	12000: 
		IF 	DetactSensor_B  AND FeedInSensor_B THEN
			uiExecutingStep := 12100;
		ELSIF NOT DetactSensor_B  AND FeedInSensor_B THEN
			uiExecutingStep := 12200;
		ELSIF DetactSensor_B  AND NOT FeedInSensor_B THEN
			uiExecutingStep := 12400;
		ELSIF NOT DetactSensor_B  AND NOT FeedInSensor_B THEN
			uiExecutingStep := 12400;
		END_IF
	12100: 	// two sensor on
			// Reversemotor unstill two sensor off
		ConveyorMotorB.M_MoveBackward();//('');
		tonMotorBReverse.IN :=TRUE;
		IF tonMotorBReverse.Q THEN
			tonMotorBReverse.IN :=FALSE;
			ConveyorMotorB.M_MotorStop();//('');
			uiExecutingStep :=12110;
		END_IF
		
	12110:	//wait conveyorA stop
		IF ConveyorMotorB.InStopped  THEN
			uiExecutingStep :=12120;
		END_IF
	12120:	//check two sensor
		IF DetactSensor_B OR FeedInSensor_B THEN
			_Error :=TRUE;
			strStatus :='PullOutConveyorB full box ,please remove';
		ELSE 
			uiExecutingStep :=12800;
		END_IF
		
	12200:	// FeedinSensor on
			//conveyor forward 
			FixCylinderB2.M_Extend();//('');
			IF  FixCylinderB2.InFrontPosition THEN
				ConveyorMotorB.M_MoveForward();// .M_Extend();//;//('');
				uiExecutingStep := 12840;
			END_IF		
	
	12400:	//two sensor off , need make sure no box in two sensor between 
			// Reverse motor to touch detactSensor , make sure no box 
			ConveyorMotorB.M_MoveBackward();//('');
			TON_betweenboxReverse.IN :=TRUE;
			IF TON_betweenboxReverse.Q THEN
				TON_betweenboxReverse.IN :=FALSE;
				ConveyorMotorB.M_MotorStop();//('');
				uiExecutingStep := 12410;
			END_IF
	12410:
			// wait motor stop
			IF ConveyorMotorB.InStopped  THEN
				uiExecutingStep :=12420;
			END_IF
	12420:	//check sensor
			IF DetactSensor_B THEN
				uiExecutingStep :=12430; // todo sth
			ELSIF NOT DetactSensor_B  THEN
				uiExecutingStep :=12800;
			END_IF 
	12430:	//reversemotor unstill sensor off
			ConveyorMotorB.M_MoveBackward();//('');
			TON_betweenboxReverse.IN :=TRUE;	//use to timeout 0.6s
			IF NOT DetactSensor_B THEN
				ConveyorMotorB.M_MotorStop();//('');
				uiExecutingStep :=12440;
			END_IF
			IF TON_betweenboxReverse.Q THEN
				_Error :=TRUE;
				strStatus :='PullOutConveyorB FeedIn full box ,please remove box';
			END_IF
	12440:	//wait motor stop
			IF ConveyorMotorB.InStopped  THEN
				uiExecutingStep :=12800;
			END_IF
			
	12800:	//BlockA forward and motorA forward
			BarrierCylinderB.M_Extend();//('');
			IF BarrierCylinderB.InFrontPosition THEN
				ConveyorMotorB.M_MoveForward();//;//('');
				uiExecutingStep :=12810;
			END_IF
	12810:	//wait box move in sensor and pressbox forward
			TON_PullOutTimeOut.IN 	:=TRUE;		//10S
			tonSensorDetectDelay.IN :=DetactSensor_B;		//100MS
			IF tonSensorDetectDelay.Q THEN
				tonSensorDetectDelay.IN :=FALSE;
				TON_PullOutTimeOut.IN 	:=FALSE;
				FixCylinderB2.M_Extend();//('');
				uiExecutingStep :=12820;
			END_IF
			IF TON_PullOutTimeOut.Q THEN
				_Error :=TRUE;
				strStatus :='PullOutConveyorA none box ,please refill box';
			END_IF
	12820:	//wait PressboxB2 forward & Blockbox backward 
			IF FixCylinderB2.InFrontPosition THEN
				BarrierCylinderB.M_Retract();//('');
				uiExecutingStep :=12830;
			END_IF
	12830:	//wait blockbox backward
			IF BarrierCylinderB.InRearPosition THEN
				uiExecutingStep :=12840;
			END_IF
	12840:	//delay sensor time
			TON_FeedInsensorADelay.IN := FeedInSensor_B ;
			IF TON_FeedInsensorADelay.Q THEN
				TON_FeedInsensorADelay.IN :=FALSE;
				ConveyorMotorB.M_MotorStop();//('');
				uiExecutingStep :=12850;
			END_IF
	12850:	//wait conveyor stop
			IF ConveyorMotorB.InStopped  THEN
				FixCylinderB1.M_Extend();//('');
				uiExecutingStep :=12860;
			END_IF
	12860:	//wait pressbox cylinder move
			IF FixCylinderB1.InFrontPosition THEN
				FixCylinderB1.M_Retract();//('');
				FixCylinderB2.M_Retract();//('');
				uiExecutingStep :=12870;
			END_IF
	12870:	//done
			IF FixCylinderB1.InRearPosition AND FixCylinderB2.InRearPosition THEN
				uiExecutingStep :=99000;
			END_IF
//	12000: 	
//			//check FeedinSensor & DetactSensor
//			tonMotorBReverse.IN :=TRUE;
//			ConveyorMotorb.M_MoveBackward();//('');				
//			IF tonMotorBReverse.Q  THEN
//					tonMotorBReverse.IN :=FALSE;
//					ConveyorMotorb.M_MotorStop();//('');
//					uiExecutingStep :=12005;
//			END_IF
//	12005: 	//check box leave sensor 
//			IF FeedInSensor_B OR DetactSensor_B THEN
//				_Error :=TRUE;
//				strStatus :='PullOutConveyorB full box ,please remove box';
//			ELSE
//				uiExecutingStep :=12010;
//			END_IF
	
//	12010:	//wait conveyorB stop
//			IF ConveyorMotorB.InStopped  THEN
//				uiExecutingStep := 12050;
//			END_IF
//	12050: 
//			//block forward 
//		BarrierCylinderB.M_Extend();//('');
//		IF BarrierCylinderB.In_FrontPosition THEN
//			uiExecutingStep := 12100;
//		END_IF
//	12100:	// motor forward & check detactsensor
//		ConveyorMotorB.M_Extend();//;//('');
//		TON_BoxArrivedDelay.IN := TRUE;
//		IF DetactSensor_B  THEN
//			uiExecutingStep := 12200;
//		END_IF
//		IF TON_BoxArrivedDelay.Q THEN
//			Status := 'SlideB FeedIn no box';
//			_Error := TRUE;
//		END_IF
//	12200:
//		tonSensorDetectDelay.IN :=TRUE;
//		IF tonSensorDetectDelay.Q THEN
//			FixCylinderB2.M_Extend();//('');
//			uiExecutingStep := 12300;
//		END_IF
//	12300:
//		tonSensorDetectDelay.IN :=FALSE;
//		BarrierCylinderB.M_Retract();//('');
//		IF BarrierCylinderB.In_RearPosition THEN
//			uiExecutingStep := 12400;
//		END_IF
//	12400:
//		TON_BoxArrivedDelay.IN := TRUE;
//		IF FeedInSensor_B THEN
//			ConveyorMotorB.M_MotorStop();//('');
//			uiExecutingStep := 12500;
//		END_IF
//		IF TON_BoxArrivedDelay.Q THEN
//			Status := 'SlideB FeedIn no box';
//			_Error := TRUE;
//		END_IF
//	12500:
//		FixCylinderB1.M_Extend();//('');
//		uiExecutingStep := 12510;
//	12510:
//		TON_BarryDelay.IN := TRUE;
//		IF TON_BarryDelay.Q THEN
//			FixCylinderB1.M_Retract();//('');
//			FixCylinderB2.M_Retract();//('');
//			uiExecutingStep := 99000;
//		END_IF
{endregion}

	50000:	//SlideA FeedIn Ext Resume step
			FixCylinderA1.M_Retract();
			FixCylinderA2.M_Retract();
			BarrierCylinderA.M_Retract();
			ConveyorMotorA.M_MotorStop();
			TON_PullOutTimeOut.IN :=FALSE;
			TON_betweenboxReverse.IN :=FALSE;
			IF FixCylinderA1.InRearPosition AND 
				FixCylinderA2.InRearPosition AND 
				BarrierCylinderA.InRearPosition AND 
				ConveyorMotorA.InStopped THEN
				_Abort :=TRUE;
			END_IF
			
    99000:
        TON_MotorStopDelay.IN := FALSE;
        _Executed             := TRUE;

END_CASE

IF _Executed THEN
    eState := STATE_DONE;
ELSIF NOT Execute THEN
    eState := STATE_RESETTING;
ELSIF _Abort OR Abort THEN
    eState := STATE_ABORTING;
ELSIF _Error THEN
	eState:=STATE_ERROR;	
END_IF
END_METHOD

METHOD  M_STATE_RESETTING
VAR_INPUT
END_VAR
CASE uiResettingStep OF
	0:
		FixCylinderA1.M_Retract();// .M_Retract();//('Resetting');
		FixCylinderA2.M_Retract();//('Resetting');
		FixCylinderB1.M_Retract();//('Resetting');
		FixCylinderB2.M_Retract();//('Resetting');
		BarrierCylinderA.M_Retract();//('Resetting');
		BarrierCylinderB.M_Retract();//('Resetting');
		uiResettingStep := 100;
	100:
		IF FixCylinderA1.InRearPosition AND
			FixCylinderA2.InRearPosition AND
			FixCylinderB1.InRearPosition AND
			FixCylinderB2.InRearPosition AND
			BarrierCylinderA.InRearPosition AND 
			BarrierCylinderB.InRearPosition THEN
			uiResettingStep := 200;
		END_IF
	200:
		ConveyorMotorA.M_MotorStop();// .M_StopMotor('Resetting');
		ConveyorMotorB.M_MotorStop();
		uiResettingStep := 300;
	300:
		IF ConveyorMotorA.InStopped AND 
			ConveyorMotorB.InStopped THEN
		//	DAS.fbStorageArea.M_InactivePulloutConveyorInternCtrl();
			uiResettingStep := 9000;
		END_IF
	9000:
		_Error :=false;
		 Error :=false;
		_ResetCompleted := TRUE;
END_CASE
IF _ResetCompleted THEN
	eState := STATE_DORMANT;
END_IF
END_METHOD

END_FUNCTION_BLOCK

// ---- Library/20_MachineUnits/22_AllocateArea/Service/FB_PullOutConveyorBtnCtrl.TcPOU
FUNCTION_BLOCK FB_PullOutConveyorBtnCtrl 
VAR_INPUT
	Input	:REFERENCE TO ST_InputTable;
	Output	:REFERENCE TO ST_OutputTable;
//	ConveyorMotorA :REFERENCE TO FB_Motor;
//	ConveyorMotorB :REFERENCE TO FB_Motor;
	Motor	:REFERENCE TO UNI_MotorList;
	
	
	bPullOutConveyorExecute	:BOOL;
	bPullOutConveyorDone	:BOOL;
	bPullOutConveyorBusy	:BOOL;
	StroageRegionMode :E_UnitMode ;
END_VAR
VAR_OUTPUT
	PullOutConveyorState :E_PullOutConveyorState;
END_VAR
VAR
	ExecutingStep	:E_PullOutConveyorState;
	bReferenceComponetIsRefed :BOOL;
	Forward_EdgeDetect	:FB_EdgeDetect;
	Backward_EdgeDetect	:FB_EdgeDetect;
END_VAR

clcUpdate();
Forward_EdgeDetect(xInput:=Input.bPullOutCV_FwdPb);
Backward_EdgeDetect(xInput :=Input.bPullOutCV_RevPb);
//IF __ISVALIDREF(BtnMoveForward) AND
//	__ISVALIDREF(BtnMoveReverse) AND
//	__ISVALIDREF(ConveyorMotorA) AND
//	__ISVALIDREF(ConveyorMotorB) THEN
	
//	bReferenceComponetIsRefed :=TRUE;
//END_IF

//IF bReferenceComponetIsRefed THEN
//	clcUpdate();
//END_IF

METHOD PRIVATE clcUpdate : BOOL
VAR_INPUT
END_VAR

CASE ExecutingStep OF
	E_PullOutConveyorState.idle:
	;
	
	E_PullOutConveyorState.AutoMode:
		M_TurnOff();
		M_TurnOff();
			IF bPullOutConveyorDone AND 
				NOT bPullOutConveyorExecute AND 
				NOT (StroageRegionMode = E_MachineMode.AUTO)  THEN
				ExecutingStep := E_PullOutConveyorState.Free;
			END_IF
	
	E_PullOutConveyorState.Free:
		M_TurnOn();
		M_TurnOn();
		IF NOT (StroageRegionMode = E_UnitMode.AUTO) AND 
				(StroageRegionMode = E_UnitMode.MANUAL) THEN
//			IF BtnMoveReverse.P_ButtonState AND BtnMoveForward.P_ButtonState THEN
			IF Input.bPullOutCV_FwdPb AND Input.bPullOutCV_RevPb THEN
//				ConveyorMotorA.M_StopMotor('');
//				ConveyorMotorB.M_StopMotor('');
				Motor.List.PullOutCV_A.M_MotorStop();
				Motor.List.PullOutCV_B.M_MotorStop();
					ELSIF Forward_EdgeDetect.xFallingEdge THEN 
						Motor.List.PullOutCV_A.M_MotorStop();
						Motor.List.PullOutCV_B.M_MotorStop();
					ELSIF Backward_EdgeDetect.xFallingEdge THEN
						Motor.List.PullOutCV_A.M_MotorStop();
						Motor.List.PullOutCV_B.M_MotorStop();
					ELSIF Input.bPullOutCV_RevPb THEN
							Motor.List.PullOutCV_A.M_MoveBackward();
							Motor.List.PullOutCV_B.M_MoveBackward();
					ELSIF Input.bPullOutCV_FwdPb  THEN
							Motor.List.PullOutCV_A.M_MoveForward();
							Motor.List.PullOutCV_B.M_MoveForward();					
			END_IF
		END_IF
END_CASE

IF (bPullOutConveyorExecute AND bPullOutConveyorBusy ) OR (StroageRegionMode = E_UnitMode.AUTO)  THEN
	ExecutingStep := E_PullOutConveyorState.AutoMode;
ELSE
	ExecutingStep := E_PullOutConveyorState.Free;
END_IF

PullOutConveyorState:=ExecutingStep;
END_METHOD

METHOD PRIVATE M_TurnOff : BOOL
VAR_INPUT
END_VAR
Output.bPullOutCV_FwdPbLamp:=FALSE;
Output.bPullOutCV_RevPbLamp:=FALSE;
END_METHOD

METHOD PRIVATE M_TurnOn : BOOL
VAR_INPUT
END_VAR
Output.bPullOutCV_FwdPbLamp:=TRUE;
Output.bPullOutCV_RevPbLamp:=TRUE;
END_METHOD

END_FUNCTION_BLOCK

// ---- Library/20_MachineUnits/22_AllocateArea/Service/FB_AllocateRobotNeedlingMove.TcPOU
FUNCTION_BLOCK FB_AllocateRobotNeedlingMove EXTENDS FB_ActionBasic
VAR_INPUT
    xExecute      : BOOL;
    xAbort        : BOOL;
    TimeOut  : LREAL := 30; // Unit : s
	MovingInfo	: ST_AllocateRobotNeedlingMoveInfo;
END_VAR
VAR_OUTPUT
    xAborted : BOOL;
    iErrorID : INT;
    ErrorMsg : T_MaxString;
END_VAR
VAR
    StateBehavior   : CBML.ETrigATo;
    uiCyclicStep    : UINT := 0;
    uiIndexLoop     : UINT;
	Coordinate		:st_Coordinate;
	fbExecuteEdgeDetect :FB_EdgeDetect;
END_VAR

THIS^.IBehaviourModel := StateBehavior;
StateBehavior(xExecute := xExecute,
              xAbort := xAbort OR fbExecuteEdgeDetect.xFallingEdge,
              udiTimeOut := LREAL_TO_UDINT( TimeOut*1000000),
              xDone => xDone,
              xBusy => xBusy,
              xError => xError,			  
              xAborted => xAborted);			  

			  
//Make sure that C# turns off execute to shut down the service
fbExecuteEdgeDetect(xInput :=xExecute);

//Error Msg
iErrorID := StateBehavior._model.iErrorID;
ErrorMsg := M_GetErrorMsg(xErrorID := iErrorID);

METHOD CleanupAction
VAR_INPUT
    xAbortProposed : BOOL;
    iErrorIDProposed: INT;
END_VAR
VAR_OUTPUT
    xComplete : BOOL := TRUE;
    xAbort: BOOL := xAbortProposed;
 	iErrorID : INT := iErrorIDProposed;
END_VAR
uiCyclicStep := 0;
END_METHOD

METHOD CyclicAction
VAR_INPUT
    itfTimingController : CBML.ITimingController;
END_VAR
VAR_OUTPUT
    xComplete : BOOL := TRUE;
    iErrorID : INT := 0;
END_VAR
VAR_INST
	
END_VAR

VAR
		bAxesCheck 		: BOOL;
	
	
END_VAR
xComplete := FALSE;

	IF arAxisCtrl_gb[AxisNo.Allocate_X].Admin.Axis.Status.Error OR
		arAxisCtrl_gb[AxisNo.Allocate_Y].Admin.Axis.Status.Error THEN
		iErrorID :=3;
	END_IF

CASE uiCyclicStep OF
    0:
		
			uiCyclicStep:=100;
		
		
	100:
			arAxisCtrl_gb[AxisNo.Allocate_X].PosMode.Position:=Coordinate.X;
			arAxisCtrl_gb[AxisNo.Allocate_Y].PosMode.Position:=Coordinate.Y;	
		
			IF arAxisCtrl_gb[AxisNo.Allocate_X].Admin.Axis.Status.Moving OR
			   arAxisCtrl_gb[AxisNo.Allocate_Y].Admin.Axis.Status.Moving OR
			   arAxisStatus_gb[AxisNo.Allocate_X].Admin._OpModeAck=E_AXIS_MODE.ModePosAbs OR
			   arAxisStatus_gb[AxisNo.Allocate_y].Admin._OpModeAck=E_AXIS_MODE.ModePosAbs THEN
			   uiCyclicStep:=200;
			END_IF
			
	200:
			bAxesCheck := TRUE;

		bAxesCheck := bAxesCheck AND	 arAxisStatus_gb[AxisNo.Allocate_x].Admin.CmdDone ;
		bAxesCheck := bAxesCheck AND	 arAxisStatus_gb[AxisNo.Allocate_y].Admin.CmdDone ;	
	
		IF bAxesCheck THEN
			 uiCyclicStep:=600;
		END_IF
	600:
		
		xComplete := TRUE;
END_CASE
END_METHOD

METHOD ExitAction
VAR_INPUT
    xAfterCleanup : BOOL;
    xInCopyCode : BOOL;
END_VAR
END_METHOD

METHOD PRIVATE M_CheckCommand : BOOL
VAR_INPUT
END_VAR
VAR_OUTPUT
	iErrorID	 : INT :=0 ;
END_VAR
VAR
	
END_VAR
IF MovingInfo.Box<0 OR MovingInfo.Box >1 OR MovingInfo.Clip<0 OR MovingInfo.Clip>3 OR MovingInfo.NeedleLocation<0 OR MovingInfo.NeedleLocation>49 THEN
	iErrorID :=2;
	M_CheckCommand := FALSE;
	RETURN;
END_IF

IF MovingInfo.Area = 'T' THEN
		
	FUN_GetNeedleCoordinates(uiLocation :=1 ,
							 uiBox:=MovingInfo.Box,
							 uiClip:=MovingInfo.Clip,
							 uiNeedleLocation:=MovingInfo.NeedleLocation,
							 NeedleCoordinate=>Coordinate);
	IF MovingInfo.Box = 1 AND (MovingInfo.Clip = 2 OR MovingInfo.Clip = 3) THEN
		M_CheckCommand := FALSE;
		iErrorID :=2;
		RETURN;
	END_IF
	IF MovingInfo.Box = 2 AND (MovingInfo.Clip = 0 OR MovingInfo.Clip = 1) THEN
		M_CheckCommand :=FALSE;
		iErrorID :=2;
		RETURN;
	END_IF
	
ELSIF 	

	MovingInfo.Area = 'Q' THEN
	FUN_GetNeedleCoordinates(uiLocation :=0 ,
							 uiBox:=MovingInfo.Box,
							 uiClip:=MovingInfo.Clip,
							 uiNeedleLocation:=MovingInfo.NeedleLocation,
							 NeedleCoordinate=>Coordinate);
	

ELSE
	iErrorID :=2;
	M_CheckCommand := FALSE;
	RETURN;
END_IF

M_CheckCommand:=TRUE;
END_METHOD

METHOD M_GetErrorMsg : T_MaxString
VAR_INPUT
	xErrorID: INT;
END_VAR

VAR
	
END_VAR
CASE xErrorID OF
	0:
		M_GetErrorMsg := 'No Error';
	1:
		M_GetErrorMsg := 'Action time out';
	2:
		M_GetErrorMsg := 'Wrong command';
	3:
		M_GetErrorMsg := 'Servo axis error';
//	4:
//		M_GetErrorMsg := 'Axis roundbelt not ready has Error';
//	5:
//		M_GetErrorMsg := 'Cylinder not ready has Error';
//	6:
//		M_GetErrorMsg := 'Axis RoundBelt has Error';
//	7:
//		M_GetErrorMsg := 'ChargeZone_Plug has Error';
//	8:
//		M_GetErrorMsg := 'TransmitCVZone_Plug has Error';
//	9:
//		M_GetErrorMsg := 'WorkZone_Plug has Error';
//	10:
//		M_GetErrorMsg := 'WorkZone_Press has Error';
END_CASE
END_METHOD

METHOD PRIVATE M_ResetAxes : BOOL
VAR_INPUT
END_VAR
VAR
	bAxesCheck :BOOL;
END_VAR
		bAxesCheck :=TRUE;
		IF arAxisCtrl_gb[AxisNo.Allocate_X].Admin.Axis.Status.Error THEN
			arAxisCtrl_gb[AxisNo.Allocate_X].Admin.ClearError:=TRUE;			
			ELSE
			arAxisCtrl_gb[AxisNo.Allocate_X].Admin.ClearError:=FALSE;	
		END_IF
		IF arAxisCtrl_gb[AxisNo.Allocate_Y].Admin.Axis.Status.Error THEN
			arAxisCtrl_gb[AxisNo.Allocate_Y].Admin.ClearError:=TRUE;			
			ELSE
			arAxisCtrl_gb[AxisNo.Allocate_Y].Admin.ClearError:=FALSE;	
		END_IF
		bAxesCheck := bAxesCheck AND NOT arAxisCtrl_gb[AxisNo.Allocate_X].Admin.ClearError ;
		bAxesCheck := bAxesCheck AND NOT arAxisCtrl_gb[AxisNo.Allocate_X].Admin.ClearError ;
		
		M_ResetAxes := bAxesCheck;
END_METHOD

METHOD ResetAction
VAR_OUTPUT
    xComplete : BOOL := TRUE;
END_VAR
uiCyclicStep := 0;
END_METHOD

METHOD StartAction
VAR_OUTPUT
    xComplete : BOOL := TRUE;
	iErrorID : INT := 0;
END_VAR
xComplete := FALSE;
uiCyclicStep := 0;

IF M_CheckCommand(iErrorID=>iErrorID) AND M_ResetAxes() THEN
	xComplete := TRUE;
END_IF
END_METHOD

END_FUNCTION_BLOCK

// ---- Library/20_MachineUnits/22_AllocateArea/Duts/F_Even.TcPOU
FUNCTION F_Even : BOOL
VAR_INPUT
	uiNumber		: UINT;
END_VAR
VAR
END_VAR

F_Even := uiNumber MOD 2 = 0;

END_FUNCTION

// ---- Library/20_MachineUnits/21_StorageArea/FB_StorageArea.TcPOU
FUNCTION_BLOCK FB_StorageArea EXTENDS FB_ModeBase_V2 IMPLEMENTS I_UnitState
VAR_INPUT
    FanucRobot : REFERENCE TO FB_FanucRobot_Basic;
    Service    : REFERENCE TO ST_StorageService;

    Cylinder : REFERENCE TO UNI_CylinderList;
    Motor    : REFERENCE TO UNI_MotorList;

    Input            : REFERENCE TO ST_InputTable;
    OutPut           : REFERENCE TO ST_OutputTable;
    Reset            : REFERENCE TO BOOL;
	Stop :  REFERENCE TO BOOL;
	bStopMem :  REFERENCE TO BOOL;
    WheelhouseSensor : REFERENCE TO UNI_HMI_WheelHouseInput;
    CurrentData      : ST_SetupPara;
END_VAR
VAR_OUTPUT
	RobotResetCMD :BOOL;
	Homed : BOOL;
END_VAR
VAR
    // Service
    fbFeedInEmptyBoxWithRobot           : FB_FeedInEmptyBoxWithRobot;
    fbReloadRoundBeltBoxWithRobot       : FB_ReloadRoundBeltBoxWithRobot;
    fbRobotRegionMove_AllocatedConveyor : FB_RobotRegionMove_AllocatedConveyor;
    fbRobotRegionMove_BufferArea        : FB_RobotRegionMove_BufferArea;
    fbRobotRegionMove_FeedInConveyor    : FB_RobotRegionMove_FeedInConveyor;
    fbRobotRegionMove_PullOutConveyor   : FB_RobotRegionMove_PullOutConveyor;
    fbRobotRegionMove_RoundBelt         : FB_RobotRegionMove_RoundBelt;
    fbRobotAbsMove                      : FB_RobotAbsMove;
    fbWareHouseWithRobotMove            : FB_WareHouseWithRobotMove;
	fbStorageHoming 					: FB_StorageHoming;
	//UpCV
    _fbDaimeterMovement   			: FB_DiameterMovement; //UpCV Internal use
    fbUpperFeedInConveyor 			: FB_UpperFeedInConveyor;
	fbAddBoxes                      : FB_AddBoxes_v2;
	fbBoxSupplyCtrl					: FB_BoxSupplyCtrl;
    RackState                       : E_RackState;
    
    // Pullout
    fbPullOutConveyorAction         : FB_PullOutConveyorAction;
    AutoPullout_Ctrl                : ST_AutoPullOutConveyorCommand;
    AutoPullout_Status              : ST_AutoPullOutConveyorSatus;
    AutoPullout_Info                : ST_PullOutConveyorInfo;
    bPulloutConveyorInternCtrl      : BOOL := FALSE;
    AutoMode_PulloutConveyor_Intern : ST_AutoPullOutConveyor; // Pullout conveyor inter
    

    // Robot abs move
    RobotAbsMoveAuto_Ctrl   : st_RobotAbsMove_Ctrl;
    RobotAbsMoveAuto_Status : st_RobotAbsMove_Status;
    RobotAbsMoveAuto_Info   : st_AutoSixAxisAbsMoveParameter;
    // Warehouse
	fbWarehouse           : FB_WareHouse;
    //========= Auto Mode Robot Warehouse Move =================
    RobotWarehouseMoveAuto_Ctrl   : st_RobotWarehouseMove_Ctrl;
    RobotWarehouseMoveAuto_Status : st_RobotWarehouseMove_Status;

    _RobotWarehouseMoveAuto_Ctrl   : st_RobotWarehouseMove_Ctrl;
    _RobotWarehouseMoveAuto_Status : st_RobotWarehouseMove_Status;

    RobotWarehouseMoveAuto_internal_Ctrl   : st_RobotWarehouseMove_Ctrl;
    RobotWarehouseMoveAuto_internal_Status : st_RobotWarehouseMove_Status;
    bWarehouseMoveInternalAccess           : BOOL := FALSE;
	// Storage homing
	StorageHoming_Execute : BOOL;
	StorageHoming_Reset : BOOL;
	StorageHoming_Abort : BOOL;
	StorageHoming_Busy : BOOL;
	StorageHoming_Done : BOOL;
	StorageHoming_Error : BOOL;
END_VAR

SUPER^();

IF __ISVALIDREF(PackTag) THEN
    eModeCommand := PackTag.Command.UnitMode;
    eStateCommand := PackTag.Command.CntrlCmd;
ELSE
    RETURN;
END_IF

ACTION A00_Service:
fbFeedInEmptyBoxWithRobot(Execute    := service.AutoMode_FeedInEmptyBoxWithRobot.Command.Execute,
                          Abort      := service.AutoMode_FeedInEmptyBoxWithRobot.Command.Abort,
                          Reset      := Reset,
                          ObjectName := 'FeedInEmptyBox with robot',
                          Busy       => service.AutoMode_FeedInEmptyBoxWithRobot.Status.Busy,
                          Done       => service.AutoMode_FeedInEmptyBoxWithRobot.Status.Done,
                          Aborted    =>,
                          Error      => service.AutoMode_FeedInEmptyBoxWithRobot.Status.Error,
                          ErrorID    =>,
                          Status     => service.AutoMode_FeedInEmptyBoxWithRobot.Status.Status,
                          UniqueErrorCode   =>,
                          Robot      := FanucRobot,
                          WareHouse  := fbWarehouse,
                          Input      := Input,
                          DiffSizeCV := Motor.List.TransmitDifferentSideCV,
						  SameSizeCV := Motor.List.TransmitSameSideCV,
                          Info := Service.AutoMode_FeedInEmptyBoxWithRobot.Info,
                          Stop := bStopMem);

fbRobotRegionMove_BufferArea(Execute	:= Service.AutoMode_RobotRegionMove_BufferArea.Command.Execute,
                             Abort 		:= Service.AutoMode_RobotRegionMove_BufferArea.Command.Abort,
                             Reset 		:= Reset,
                             ObjectName	:= 'RobotRegionMove_BufferArea',
                             Busy    => Service.AutoMode_RobotRegionMove_BufferArea.Status.Busy,
                             Done    => Service.AutoMode_RobotRegionMove_BufferArea.Status.Done,
                             Aborted =>,
                             Error   => Service.AutoMode_RobotRegionMove_BufferArea.Status.Error,
                             ErrorID =>,
                             Status  => Service.AutoMode_RobotRegionMove_BufferArea.Status.Status,
							 UniqueErrorCode	=>,
                             Robot 	:= FanucRobot,
                             Info 	:= Service.AutoMode_RobotRegionMove_BufferArea.Info,
                             Stop 	:= bStopMem);

fbPullOutConveyorAction(Execute          := (*AutoPullout_Ctrl.Execute*) ,
                        Abort            := AutoPullout_Ctrl.Abort,
                        Reset            := Reset,
                        ObjectName       := 'fbPullOutConveyorAction',
                        Busy             => AutoPullout_Status.Busy,
                        Done             => AutoPullout_Status.Done,
                        Aborted          =>,
                        Error            => AutoPullout_Status.Error,
                        ErrorID          =>,
                        Status           => AutoPullout_Status.Status,
                        UniqueErrorCode  =>,
                        FixCylinderA1    := Cylinder.List.fbPullOutCV_AsidePress1,
                        FixCylinderA2    := Cylinder.List.fbPullOutCV_AsidePress2,
                        FixCylinderB1    := Cylinder.List.fbPullOutCV_BsidePress1,
                        FixCylinderB2    := Cylinder.List.fbPullOutCV_BsidePress2,
                        BarrierCylinderA := Cylinder.List.fbPullOutCV_AsideBlock,
                        BarrierCylinderB := Cylinder.List.fbPullOutCV_BsideBlock,
                        ConveyorMotorA   := Motor.List.PullOutCV_A,
                        ConveyorMotorB   := Motor.List.PullOutCV_B,
                        INPUT            := INPUT,
                        PullOutInfo      := AutoPullout_Info);

fbUpperFeedInConveyor(Execute             := Service.AutoMode_UpperFeedInConveyor.Command.Execute,
                      Abort               := Service.AutoMode_UpperFeedInConveyor.Command.Abort,
                      Reset               := Reset,
                      ObjectName          := 'Storage_UpperFeedInConveyor',
                      Busy                => Service.AutoMode_UpperFeedInConveyor.Status.Busy,
                      Done                => Service.AutoMode_UpperFeedInConveyor.Status.Done,
                      Aborted             =>,
                      Error               => Service.AutoMode_UpperFeedInConveyor.Status.Error,
                      ErrorID             =>,
                      Status              =>,
                      UniqueErrorCode     =>,
                      _fbDiameterMovement := THIS^._fbDaimeterMovement,
                      Cylinder            := Cylinder,
                      Motor               := Motor,
                      Input               := Input,
                      OutPut              := OutPut,
                      Info                := Service.AutoMode_UpperFeedInConveyor.Info,
                      AddingBox           :=,
                      FeedBack            => Service.AutoMode_UpperFeedInConveyor.FeedBack,
					  _bForceUpperCV_Use   =>	);

_fbDaimeterMovement(Execute         :=,
                    Abort           :=,
                    Reset           :=,
                    ObjectName      :=,
                    Busy            =>,
                    Done            =>,
                    Aborted         =>,
                    Error           =>,
                    ErrorID         =>,
                    Status          =>,
                    UniqueErrorCode =>,
                    bContinue       :=,
                    Cylinder        := Cylinder,
                    PickDone        =>);

fbWarehouse(Motors           := Motor,
            WheelhouseSensor := WheelhouseSensor);

fbAddBoxes(Execute                   := Service.AutoMode_AddBoxes.Command.Execute,
           Abort                     := Service.AutoMode_AddBoxes.Command.Abort,
           Reset                     := Reset,
           ObjectName                := 'Storage_AddBoxes',
           Busy                      => Service.AutoMode_AddBoxes.Status.Busy,
           Done                      => Service.AutoMode_AddBoxes.Status.Done,
           Aborted                   =>,
           Error                     => Service.AutoMode_AddBoxes.Status.Error,
           ErrorID                   =>,
           Status                    =>,
           UniqueErrorCode           =>,
           Cylinder                  := Cylinder,
           Motor                     := Motor,
           Input                     := Input,
           OutPut                    := OutPut,
           CurrentData               := CurrentData,
           ERackState                := RackState,
           bClearInterventionRequest :=,
           InterventionRequest       => Service.AutoMode_AddBoxes.Status.InterventionRequest,
           FeedingBoxes              => Service.AutoMode_AddBoxes.Status.FeedingBoxes,
			_bForceUpperCV_Use 		:= fbUpperFeedInConveyor._bForceUpperCV_Use);

fbBoxSupplyCtrl(Execute           := TRUE,
                Abort             :=,
                Reset             :=reset,
                ObjectName        :=,
                Busy              =>,
                Done              =>,
                Aborted           =>,
                Error             =>,
                ErrorID           =>,
                Status            =>,
                UniqueErrorCode   =>,
                Cylinder          := Cylinder,
                CurrentData       := CurrentData,
                Input             := Input,
                Output            := OutPut,
                StroageRegionMode := eModeCurrent,
                bAddsBoxRequest   := Service.AutoMode_AddBoxes.Status.InterventionRequest,
                AddBoxes_Status   := Service.AutoMode_AddBoxes.Status,
                AddBoxes_Ctrl     := Service.AutoMode_AddBoxes.Command,
				AxisRackMotorBTNHomeRequest=>,
                RackState         => RackState);

fbRobotRegionMove_FeedInConveyor(Execute 	:= Service.AutoMode_RobotRegionMove_FeedInConveyor.Command.Execute,
                                 Abort 		:= Service.AutoMode_RobotRegionMove_FeedInConveyor.Command.Abort,
                                 Reset      := Reset,
                                 ObjectName := 'Storage Robot FeedIn CV',
                                 Busy       => Service.AutoMode_RobotRegionMove_FeedInConveyor.Status.Busy,
                                 Done 		=> Service.AutoMode_RobotRegionMove_FeedInConveyor.Status.Done,
                                 Aborted	=>,
                                 Error   	=> Service.AutoMode_RobotRegionMove_FeedInConveyor.Status.Error,
                                 ErrorID 	=>,
                                 Status  	=> Service.AutoMode_RobotRegionMove_FeedInConveyor.Status.Status,
                                 UniqueErrorCode =>,
                                 Robot           := FanucRobot,
                                 LowerConveyor   := Motor.List.LowCV,
                                 Input           := Input,
                                 //								 F1SensorOfUpperConveyor :=Input.bUpCV_BoxArrived_Sensor,
                                 //								 Input.bUpCV_Block1Detect_Sensor := Input.bUpCV_Block1Detect_Sensor ,
                                 Info := Service.AutoMode_RobotRegionMove_FeedInConveyor.Info,
                                 Stop :=bStopMem);

fbRobotRegionMove_AllocatedConveyor(Execute 	:= Service.AutoMode_RobotRegionMove_AllocatedConveyor.Command.Execute,
                                    Abort 		:= Service.AutoMode_RobotRegionMove_AllocatedConveyor.Command.Abort,
                                    Reset  		:= Reset,
                                    ObjectName 	:= ' Storage Robot Transmit CV',
                                    Busy       	=> Service.AutoMode_RobotRegionMove_AllocatedConveyor.Status.Busy,
                                    Done 		=> Service.AutoMode_RobotRegionMove_AllocatedConveyor.Status.Done,
                                    Aborted 	=>,
                                    Error   	=> Service.AutoMode_RobotRegionMove_AllocatedConveyor.Status.Error,
                                    ErrorID 	=>,
                                    Status  	=> Service.AutoMode_RobotRegionMove_AllocatedConveyor.Status.Status,
                                    UniqueErrorCode =>,
                                    Robot           := FanucRobot,
                                    DifferenceCV    := Motor.List.TransmitDifferentSideCV,
                                    SamesizeCV      := Motor.List.TransmitSameSideCV,
                                    cylinder        := Cylinder,
                                    //	SameSizeFullSensor:= , 
                                    Input := Input,
                                    Info := service.AutoMode_RobotRegionMove_AllocatedConveyor.Info,
                                    Stop :=bStopMem);


fbRobotRegionMove_PullOutConveyor(Execute 	:=Service.AutoMode_RobotRegionMove_PullOutConveyor.Command.Execute,
                                  Abort 	:=Service.AutoMode_RobotRegionMove_PullOutConveyor.Command.Abort,
                                  Reset     := Reset,
                                  ObjectName:= 'Storage Robot PulloutCV',
                                  Busy      => Service.AutoMode_RobotRegionMove_PullOutConveyor.Status.Busy,
                                  Done 		=> Service.AutoMode_RobotRegionMove_PullOutConveyor.Status.Done,
                                  Aborted 	=>,
                                  Error   	=> Service.AutoMode_RobotRegionMove_PullOutConveyor.Status.Error,
                                  ErrorID 	=>,
                                  Status  	=> Service.AutoMode_RobotRegionMove_PullOutConveyor.Status.Status,
                                  UniqueErrorCode =>,
                                  Robot           := FanucRobot,
                                  PullOutConveyor := fbPullOutConveyorAction,
                                  Info := Service.AutoMode_RobotRegionMove_PullOutConveyor.Info,
                                  Stop :=bStopMem);

fbRobotAbsMove(Execute         := Service.AutoMode_RobotAbsMove.HandShake.Execute,
               Abort           :=,
               Reset           := Reset,
               ObjectName      := 'Storage robot abs move',
               Busy            => Service.AutoMode_RobotAbsMove.HandShake.Busy,
               Done            => Service.AutoMode_RobotAbsMove.HandShake.Done,
               Aborted         =>,
               Error           => Service.AutoMode_RobotAbsMove.HandShake.Error,
               ErrorID         =>,
               Status          =>,
               UniqueErrorCode =>,
               Robot           := FanucRobot,
               LowerConveyor   := Motor.List.LowCV,
               Info            := Service.AutoMode_RobotAbsMove,
               Input 		:= Input,
               Stop :=bStopMem);

fbRobotRegionMove_RoundBelt(Execute := Service.AutoMode_RobotRegionMove_RoundBelt.Command.Execute,
                            Abort   := Service.AutoMode_RobotRegionMove_RoundBelt.Command.Abort,
                            Reset   := Reset,
                            ObjectName:= 'Storage robot  RegionMove roundbelt',
                            Busy    => Service.AutoMode_RobotRegionMove_RoundBelt.Status.Busy,
                            Done    => Service.AutoMode_RobotRegionMove_RoundBelt.Status.Done,
                            Aborted =>,
                            Error   => Service.AutoMode_RobotRegionMove_RoundBelt.Status.Error,
                            ErrorID =>,
                            Status 	=> Service.AutoMode_RobotRegionMove_RoundBelt.Status.Status,
                            UniqueErrorCode =>,
                            Robot 		:= FanucRobot,
                            RoundBelt 	:= DAS_CoreSys.MachineControl.fbAllocateArea.RoundBeltControl,
							Input 		:= Input,
                            Info 		:= Service.AutoMode_RobotRegionMove_RoundBelt.Info,
                            Stop 		:=bStopMem);

fbReloadRoundBeltBoxWithRobot(Execute	:= Service.AutoMode_ReloadRoundBeltBoxWithRobot.Command.Execute,
                              Abort 	:= Service.AutoMode_ReloadRoundBeltBoxWithRobot.Command.Abort,
                              Reset 	:= Reset,
                              ObjectName:= 'Storage robot reload roundbelt',
                              Busy    => Service.AutoMode_ReloadRoundBeltBoxWithRobot.Status.Busy,
                              Done    => Service.AutoMode_ReloadRoundBeltBoxWithRobot.Status.Done,
                              Aborted =>,
                              Error   => Service.AutoMode_ReloadRoundBeltBoxWithRobot.Status.Error,
                              ErrorID =>,
                              Status  => Service.AutoMode_ReloadRoundBeltBoxWithRobot.Status.Status,
                              UniqueErrorCode =>,
                              Robot 	:= FanucRobot,
                              RoundBelt := DAS_CoreSys.MachineControl.fbAllocateArea.RoundBeltControl,
                              WareHouse := fbWarehouse,
                              Input 	:= Input,
                              Info 		:= Service.AutoMode_ReloadRoundBeltBoxWithRobot.Info,
                              Stop 		:= bStopMem);
//============================ Auto Mode Robot Warehouse Move =============================
IF NOT bWarehouseMoveInternalAccess THEN
    _RobotWarehouseMoveAuto_Ctrl := RobotWarehouseMoveAuto_Ctrl;
    RobotWarehouseMoveAuto_Status := _RobotWarehouseMoveAuto_Status;
ELSE
    _RobotWarehouseMoveAuto_Ctrl := RobotWarehouseMoveAuto_internal_Ctrl;
    RobotWarehouseMoveAuto_internal_Status := _RobotWarehouseMoveAuto_Status;
END_IF

(*M_RobotWarehouseMove(
        bExecute  := Service.AutoMode_RobotWarehouseMove.HandShake.Execute,
        bReset    := Service.AutoMode_RobotWarehouseMove.HandShake.Reset,
        bAbort    := FALSE,
        bOccupied := FALSE,
        eMode     := E_MachineMode.Auto,
        bBusy     => Service.AutoMode_RobotWarehouseMove.HandShake.Busy,
        bDone     => Service.AutoMode_RobotWarehouseMove.HandShake.Done,
        bError    => Service.AutoMode_RobotWarehouseMove.HandShake.Error);*)
fbWareHouseWithRobotMove(
	Execute:= Service.AutoMode_WarehouseMotoWithRobotMove.HandShake.Execute, 
	Abort:= , 
	Reset:= Reset, 
	ObjectName:= 'storage Robot Warehouse move', 
	Busy=> Service.AutoMode_WarehouseMotoWithRobotMove.HandShake.Busy, 
	Done=> Service.AutoMode_WarehouseMotoWithRobotMove.HandShake.Done, 
	Aborted=> , 
	Error=> Service.AutoMode_WarehouseMotoWithRobotMove.HandShake.Error, 
	ErrorID=> , 
	Status=> , 
	UniqueErrorCode=> , 
	Robot:= FanucRobot, 
	WareHouse:= fbWarehouse, 
	Info:= Service.AutoMode_WarehouseMotoWithRobotMove, 
	Stop:= bStopMem);
	
fbStorageHoming(
	xDone=> , 
	xBusy=> , 
	xError=> , 
	xExecute:= , 
	xAbort:= , 
	Cylinder:= Cylinder, 
	Motor:= Motor, 
	FanucRobot:= FanucRobot,
	Homed := Homed,
	xAborted=> , 
	iErrorID=> , 
	ErrorMsg=> , 
	RobotResetCMD=> RobotResetCMD,
	RackMotorHomeRequest=>);
END_ACTION

METHOD M_Aborted
M_StateComplete();
END_METHOD

METHOD M_AbortHoming
VAR_INPUT
END_VAR
StorageHoming_Abort := TRUE;
END_METHOD

METHOD M_Aborting
M_StateComplete();
END_METHOD

METHOD M_ActivePulloutConveyorInternCtrl : BOOL
VAR_INPUT
END_VAR
bPulloutConveyorInternCtrl := TRUE;

M_ActivePulloutConveyorInternCtrl := TRUE; // Method end
END_METHOD

METHOD M_ActivePulloutConveyorInternCtrl_1 : BOOL
VAR_INPUT
END_VAR
bPulloutConveyorInternCtrl := TRUE;

M_ActivePulloutConveyorInternCtrl_1 := TRUE; // Method end
END_METHOD

METHOD M_AutoPullOutConveyorActive : BOOL
VAR_INPUT
END_VAR
IF eModeCurrent = E_UnitMode.AUTO AND NOT bPulloutConveyorInternCtrl THEN
    // GVL -> AutoSimpleAllocate_Ctrl
    AutoPullout_Ctrl.Execute := service.AutoMode_PullOutConveyor.Command.Execute;
    AutoPullout_Ctrl.Abort   := service.AutoMode_PullOutConveyor.Command.Abort;
    AutoPullout_Ctrl.Reset   := service.AutoMode_PullOutConveyor.Command.Reset OR Reset;
	M_LoadingPullOutConveyorData();
ELSIF eModeCurrent = E_UnitMode.AUTO AND bPulloutConveyorInternCtrl THEN
    AutoPullout_Ctrl.Execute := AutoMode_PulloutConveyor_Intern.Command.Execute;
    AutoPullout_Ctrl.Abort   := AutoMode_PulloutConveyor_Intern.Command.Abort;
    AutoPullout_Ctrl.Reset   := AutoMode_PulloutConveyor_Intern.Command.Reset OR Reset;
	M_LoadingPullOutConveyorData();
ELSE
    AutoPullout_Ctrl.Execute := FALSE;
    AutoPullout_Ctrl.Abort   := FALSE;
    AutoPullout_Ctrl.Reset   := FALSE;
END_IF

// AutoSimpleAllocate_Status - > GVL
service.AutoMode_PullOutConveyor.Status.Busy := AutoPullout_Status.Busy;
service.AutoMode_PullOutConveyor.Status.Done := AutoPullout_Status.Done;
service.AutoMode_PullOutConveyor.Status.Error:= AutoPullout_Status.Error;
AutoMode_PulloutConveyor_Intern.Status.Busy := AutoPullout_Status.Busy;
AutoMode_PulloutConveyor_Intern.Status.Done:= AutoPullout_Status.Done;
AutoMode_PulloutConveyor_Intern.Status.Error:= AutoPullout_Status.Error;
END_METHOD

METHOD M_Clearing
M_StateComplete();
END_METHOD

METHOD M_Complete
M_StateComplete();
END_METHOD

METHOD M_Completing
M_StateComplete();
END_METHOD

METHOD M_Execute
CASE eModeCurrent OF
	E_UnitMode.Manual:
	
	E_UnitMode.Auto:
END_CASE
A00_Service();
//M_StateComplete();
END_METHOD

METHOD M_Held
M_StateComplete();
END_METHOD

METHOD M_Holding
//fbRobotRegionMove_BufferArea.Stop := TRUE;
M_StateComplete();
END_METHOD

METHOD M_Idle
M_StateComplete();
END_METHOD

METHOD M_InactivePulloutConveyorInternCtrl : BOOL
VAR_INPUT
END_VAR
bPulloutConveyorInternCtrl := FALSE;

M_InactivePulloutConveyorInternCtrl := TRUE; // Method end
END_METHOD

METHOD PRIVATE M_LoadingPullOutConveyorData : BOOL
VAR_INPUT
END_VAR
IF eModeCurrent = E_UnitMode.Manual AND NOT bPulloutConveyorInternCtrl THEN
    AutoPullout_Info := Service.AutoMode_PullOutConveyor .PullOutConveyorInfo;
ELSIF eModeCurrent = E_UnitMode.Auto AND bPulloutConveyorInternCtrl THEN
    AutoPullout_Info := AutoMode_PulloutConveyor_Intern.PullOutConveyorInfo;
END_IF

M_LoadingPullOutConveyorData := TRUE; // Method end
END_METHOD

METHOD M_ResetSlideA_FeedIn : BOOL
VAR_INPUT
END_VAR
AutoMode_PulloutConveyor_Intern.Command.Execute := FALSE;

M_ResetSlideA_FeedIn := FALSE;
END_METHOD

METHOD M_ResetSlideB_FeedIn : BOOL
VAR_INPUT
END_VAR
AutoMode_PulloutConveyor_Intern.Command.Execute := FALSE;

M_ResetSlideB_FeedIn := FALSE;
END_METHOD

METHOD M_ResetSlides_FeedOut : BOOL
VAR_INPUT
END_VAR
AutoMode_PulloutConveyor_Intern.Command.Execute := FALSE;

M_ResetSlides_FeedOut := FALSE;
END_METHOD

METHOD M_Resetting
M_StateComplete();
END_METHOD

METHOD M_RobotWarehouseMove : BOOL
VAR_INPUT
	bExecute			: BOOL;
	bReset				: BOOL;
	bAbort				: BOOL;
	bOccupied			: BOOL;
	eMode				: E_MachineMode;
END_VAR

VAR_OUTPUT
	bBusy				: BOOL;
	bDone				: BOOL;
	bError				: BOOL;
END_VAR
CASE eMode OF
	E_MachineMode.MANUAL:
//		RobotWarehouseMoveManual_Ctrl.bExecute := bExecute;
//		RobotWarehouseMoveManual_Ctrl.bReset := bReset;
//		RobotWarehouseMoveManual_Ctrl.bAbort := E_Stop;
//		RobotWarehouseMoveManual_Ctrl.bOccupied := bOccupied;
		
//		bBusy := RobotWarehouseMoveManual_Status.bBusy;
//		bDone := RobotWarehouseMoveManual_Status.bDone;
//		bError := RobotWarehouseMoveManual_Status.bError;
		
	E_MachineMode.AUTO:
//		RobotWarehouseMoveAuto_Ctrl.bExecute := bExecute;
//		RobotWarehouseMoveAuto_Ctrl.bReset := bReset;
//		RobotWarehouseMoveAuto_Ctrl.bAbort := E_Stop;
//		RobotWarehouseMoveAuto_Ctrl.bOccupied := bOccupied;
		
//		bBusy := RobotWarehouseMoveAuto_Status.bBusy;
//		bDone := RobotWarehouseMoveAuto_Status.bDone;
//		bError := RobotWarehouseMoveAuto_Status.bError;
END_CASE
END_METHOD

METHOD M_RobotWarehouseMove_1 : BOOL
VAR_INPUT
	bExecute			: BOOL;
	bReset				: BOOL;
	bAbort				: BOOL;
	bOccupied			: BOOL;
	eMode				: E_MachineMode;
END_VAR

VAR_OUTPUT
	bBusy				: BOOL;
	bDone				: BOOL;
	bError				: BOOL;
END_VAR
CASE eMode OF
	E_MachineMode.MANUAL:
//		RobotWarehouseMoveManual_Ctrl.bExecute := bExecute;
//		RobotWarehouseMoveManual_Ctrl.bReset := bReset;
//		RobotWarehouseMoveManual_Ctrl.bAbort := E_Stop;
//		RobotWarehouseMoveManual_Ctrl.bOccupied := bOccupied;
		
//		bBusy := RobotWarehouseMoveManual_Status.bBusy;
//		bDone := RobotWarehouseMoveManual_Status.bDone;
//		bError := RobotWarehouseMoveManual_Status.bError;
		
	E_MachineMode.AUTO:
//		RobotWarehouseMoveAuto_Ctrl.bExecute := bExecute;
//		RobotWarehouseMoveAuto_Ctrl.bReset := bReset;
//		RobotWarehouseMoveAuto_Ctrl.bAbort := E_Stop;
//		RobotWarehouseMoveAuto_Ctrl.bOccupied := bOccupied;
		
//		bBusy := RobotWarehouseMoveAuto_Status.bBusy;
//		bDone := RobotWarehouseMoveAuto_Status.bDone;
//		bError := RobotWarehouseMoveAuto_Status.bError;
END_CASE
END_METHOD

METHOD M_StartHoming
VAR_INPUT
END_VAR
fbStorageHoming.xExecute := TRUE;
END_METHOD

METHOD M_Starting
M_StateComplete();
END_METHOD

METHOD M_StartSlideA_FeedIn : BOOL
VAR_INPUT
END_VAR
AutoMode_PulloutConveyor_Intern.PullOutConveyorInfo.CommandType :=E_PullOutConveyorCommandType.SlideA_FeedIn_Ext;

AutoMode_PulloutConveyor_Intern.Command.Execute := TRUE;

M_StartSlideA_FeedIn := TRUE; // Method end
END_METHOD

METHOD M_StartSlideA_FeedOut : BOOL
VAR_INPUT
	ReverseTimeDelay : Time;
END_VAR
AutoMode_PulloutConveyor_Intern.PullOutConveyorInfo.CommandType :=E_PullOutConveyorCommandType.SlideA_FeedOut_Ext;
AutoMode_PulloutConveyor_Intern.PullOutConveyorInfo.ConveyorReverseTime :=ReverseTimeDelay;
AutoMode_PulloutConveyor_Intern.Command.Execute := TRUE;

M_StartSlideA_FeedOut := TRUE; // Method end
END_METHOD

METHOD M_StartSlideB_FeedIn : BOOL
VAR_INPUT
END_VAR
AutoMode_PulloutConveyor_Intern.PullOutConveyorInfo.CommandType :=E_PullOutConveyorCommandType.SlideB_FeedIn_Ext;

AutoMode_PulloutConveyor_Intern.Command.Execute := TRUE;

M_StartSlideB_FeedIn := TRUE; // Method end
END_METHOD

METHOD M_StartSlideB_FeedOut : BOOL
VAR_INPUT
	ReverseTimeDelay : Time;
END_VAR
AutoMode_PulloutConveyor_Intern.PullOutConveyorInfo.CommandType :=E_PullOutConveyorCommandType.SlideB_FeedOut_Ext;
AutoMode_PulloutConveyor_Intern.PullOutConveyorInfo.ConveyorReverseTime :=ReverseTimeDelay;
AutoMode_PulloutConveyor_Intern.Command.Execute := TRUE;

M_StartSlideB_FeedOut := TRUE; // Method end
END_METHOD

METHOD M_StopHoming
VAR_INPUT
END_VAR
fbStorageHoming.xExecute := False;
END_METHOD

METHOD M_Stopped
//fbRobotRegionMove_BufferArea.Stop := FALSE;
M_StateComplete();
END_METHOD

METHOD M_Stopping

M_StateComplete();
END_METHOD

METHOD M_Suspended
M_StateComplete();
END_METHOD

METHOD M_Suspending
M_StateComplete();
END_METHOD

METHOD M_Undefined
M_StateComplete();
END_METHOD

METHOD M_Unholding
//fbRobotRegionMove_BufferArea.Stop := FALSE;
M_StateComplete();
END_METHOD

METHOD M_Unsuspending
M_StateComplete();
END_METHOD

END_FUNCTION_BLOCK

// ---- Library/10_Machine/19_Device/FanucRobot/FB_FanucRobot_Basic.TcPOU
FUNCTION_BLOCK FB_FanucRobot_Basic IMPLEMENTS IBasicElement
VAR_INPUT
    Estop  : BOOL; // PLC ->send to Robot E-Stop
    OpMode : E_FanucRobotOpMode := RSR01; // Select Fanuc robot prog RSR1~RSR3
    Start  : BOOL;
    Reset  : BOOL; // Reset Fanuc Robot prog
    Hold   : BOOL; // PLC - > Robot send hold command
	ManualCtrl : REFERENCE TO ST_Manual_FanucRobot;
END_VAR

VAR_OUTPUT
    qEnable       : BOOL;
    qFault        : BOOL;
    E_Stop_Output : BOOL; // Touch pannel's E-Stop has been trig;
    Halt          : BOOL; // True : Robot in helt state.
    Error         : BOOL; // True : Robot has error
    ErrorID       : UDINT; // Error ID output
	ErrMsg 		  : T_MaxString;	  
END_VAR

VAR
    // Slot1
    _rawIn_UI AT %I*  : ARRAY[0..3] OF BYTE; // UI : Fanuc robot default input rawdate
    _rawOut_UO AT %Q* : ARRAY[0..3] OF BYTE; // UO : Fanuc robot default output rawdate
    // Slot2
    _rawIn_DI AT %I*           : ARRAY[0..31] OF BYTE; // DI : user define input rawdate
    _rawOut_DO AT %Q*          : ARRAY[0..31] OF BYTE; // DO : user define output rawdate
    _EIPConnectionState AT %I* : UINT; // EIP connection State (EL6652 to Fanuc Robot)
    _FanucEIPState AT %I*      : UINT; // EIP module links to FanucRobot state
    _UI1                       : ST_FanucUI1; // Fanuc Robot default Input
    _UO1                       : ST_FanucUO1; // Fanuc Robot default Output
    _DO1                       : ST_Fanuc_WarehouseHandshake; // Fanuc robot program's handshake for clampA warehouse pick / place box
    _DO2                       : ST_Fanuc_WarehouseHandshake; // Fanuc robot program's handshake for clampB warehouse pick / place box
    _DO3                       : ST_Fanuc_AbsMove; // Fanuc robot program's handshake for clampA to target area pick / place box
    _DO4                       : ST_Fanuc_AbsMove; // Fanuc robot program's handshake for clampB to target area pick / place box
    _DO5                       : ST_Fanuc_GeneralCommand; // Fanuc robot program's handshake for general control
    _DO6                       : ST_ReadWriteParaCmd; // Fanuc robot Read/Write parameter command 
    _DO7                       : INT; // Write process X position offset
    _DO8                       : INT; // Write process Y position offset
    _DO9                       : INT; // Write process Z position offset
    _DO10                      : INT; // Write process W position offset
    _DO11                      : INT; // Write process P position offset
    _DO12                      : INT; // Write process R position offset
    _Do13                      : INT; // Write process Area index
    _Do14                      : INT; // Write process Address index
    _Do15                      : INT; // Write process Layer index
    _DO16                      : INT; // Write process Slide index
    _DO17                      : ST_CCD_ZoneUse; // Set Robot use ccd or not.
    _DI1                       : ST_Fanuc_Status; // Fanuc robot program's handshake for process status
    _DI2                       : INT; // Readprocess X position offset
    _DI3                       : INT; // Read process Y position offset
    _DI4                       : INT; // Read process Z position offset
    _DI5                       : INT; // Read process W position offset
    _DI6                       : INT; // Read process P position offset
    _DI7                       : INT; // Read process R position offset
    _DI8                       : INT; // Read process Area index
    _DI9                       : INT; // Read process Address index
    _DI10                      : INT; // Read Process Layer index
    _DI11                      : INT; // Read Process Slide index
    _DI12                      : ST_ReadWriteParaStatus; // Read/Write process Status
    _VelocityCommand           : ST_IntToBool; // Robot coordenate velocity
    // Prog inside
    eState               : E_MethodStatus_Basic;
    uiRobotExecutingStep : UINT;
    uiRobotResettingStep : UINT;
    _Error               : BOOL;
    _Abort               : BOOL;
    TON_Restart_delay    : TON;
    TON_Reset_delay      : TON;
    Rtrig_RebootRobot    : R_TRIG;
    //fbReadSingleOffsetData  : FB_ReadSingleOffsetData;
    //fbWriteSingleOffsetData : FB_WriteSingleOffsetData;
    _Status               : T_MaxString;
    _eOpMode              : E_FanucRobotOpMode;
    _ModeChanging         : BOOL;
    _Completed            : BOOL;
    _ModeChanged          : BOOL;
    _uiRSR01_Step         : UINT;
    _uiRSR02_Step         : UINT;
    _uiRSR03_Step         : UINT;
    _RetryCount           : INT := 0;
    Ton_SetProgTimeOut    : TON; // This timer is used to counting the time to switch FanucRobot prog over range.
    _RSR1_Ready           : BOOL; // Fanuc Robot running in RSR1 prog, allow to Warehouse or AbsMove command.
    _RSR2_Completed       : BOOL; // Fanuc Robot finished the homing prog.
    _RSR3_Ready           : BOOL; // Fanuc Robot ready to work.
    TON_ResetFixDelay     : TON;
    Ton_RSR_SwitchDelay   : TON; // This timer is used to counting the time to switch rsr prog
    ErrorCode             : ST_IntToBool; // This value is which read from fanuc robot.
    Ton_START_SwitchDelay : TON; // This timer is used to counting the time to switch Start signal, Fanuc process need on 0.3s and off
END_VAR

VAR CONSTANT
    RetryMaxTimes   : INT  := 3;
    tSwitchProgTime : TIME := T#1S;
    tResetFixTime   : TIME := T#0.3S;
END_VAR

// Active base units.
A00_BaseUnit();
// Active mode controller
A10_ModeControl();
// Active state controller
A20_ErrorHandle();

Update();

ACTION A00_BaseUnit:
Ton_SetProgTimeOut(PT := tSwitchProgTime);
TON_Restart_delay(PT := T#1S); // Fanuc Robot need IMSTP on over 1s
TON_Reset_delay(PT := T#1S);
TON_ResetFixDelay(PT := tResetFixTime);
Ton_RSR_SwitchDelay(PT := T#0.3S);
Ton_START_SwitchDelay(PT := T#0.4S); // Fanuc Robot need on 0.3s and then set off
E_Stop_Output := _DI12.E_Stop;
END_ACTION

ACTION A10_ModeControl:
CASE _eOpMode OF
	E_FanucRobotOpMode.RSR01:
		M_ControlRSR01(bCompleted=> _Completed, ModeChanging=> _ModeChanging, ModeChanged=> _ModeChanged);
	E_FanucRobotOpMode.RSR02:
		M_ControlRSR02(bCompleted=> _Completed, ModeChanging=> _ModeChanging, ModeChanged=> _ModeChanged);
END_CASE
END_ACTION

ACTION A20_ErrorHandle:
ErrMsg := _Status;
END_ACTION

ACTION A20_StateControl:
TON_Restart_delay(PT := T#0.5S);
TON_Reset_delay(PT:=T#0.5S);
CASE eState OF
    E_MethodStatus_Basic.STATE_DORMANT:
        Enable(FALSE);
        M_Reset(FALSE);
        uiRobotExecutingStep := 0;
        uiRobotResettingStep := 0;

		IF _eOpMode = RSR01 OR _eOpMode = RSR02 OR _eOpMode = RSR03 THEN
			eState := E_MethodStatus_Basic.STATE_EXECUTING;
		END_IF
    E_MethodStatus_Basic.STATE_EXECUTING:
        CASE uiRobotExecutingStep OF
            0:
                Enable(iTrigger := TRUE);
                M_Reset(iTrigger := TRUE);
				TON_Reset_delay.in := TRUE;
                IF TON_Reset_delay.Q THEN
                    uiRobotExecutingStep := 100;
                END_IF
            100:
                M_Reset(iTrigger := FALSE);
				TON_Reset_delay.IN := FALSE;
                IF _UO1.UO01_CmdEnabled AND _UO1.UO02_SystemReady THEN
					_VelocityCommand.nInt := 1;
                    uiRobotExecutingStep := 200;
                END_IF
            200:
				// Clear Fanuc robot's action
				GVL_ADS.AutoMode_WarehouseMotoWithRobotMove.HandShake.Execute := FALSE;
				GVL_ADS.AutoMode_RobotAbsMove.HandShake.Execute := FALSE;
				_DO1.bExecute := FALSE; // Warehouse with robot clampA
				_DO2.bExecute := FALSE; // Warehouse with robot clampB
				_DO3.bExecute := FALSE; // AbsMove with robot clampA
				_DO4.bExecute := FALSE; // AbsMove with robot clampB
				uiRobotExecutingStep := 250;
			300:
				// Switch RSR3 and read all of offset data
				GVL_ADS.FanucRobot_ReadAllOffsetData.Command.Execute := TRUE;
				IF GVL_ADS.FanucRobot_ReadAllOffsetData.Status.Done THEN
					uiRobotExecutingStep := 400;
				ELSIF GVL_ADS.FanucRobot_ReadAllOffsetData.Status.Error THEN
					_Error := TRUE;
					_Status := 'Read All offset data failue';
				END_IF
			400:
                _UI1.UI09_RSR1 := TRUE;

                IF _UO1.UO11_ACK1 THEN
                    uiRobotExecutingStep := 500;
                END_IF
            500:
                _UI1.UI09_RSR1       := FALSE;
				_VelocityCommand.nInt := 30;
                uiRobotExecutingStep := 600;
            600: // Wait command
				_DO5.ClampA_Close :=  GVL_ADS.FanucRobot_General.Command.ClampA_Close;
				_DO5.ClampA_Open := GVL_ADS.FanucRobot_General.Command.ClampA_Open;
				_DO5.ClampB_Close := GVL_ADS.FanucRobot_General.Command.ClampB_Close;
				_DO5.ClampB_Open := GVL_ADS.FanucRobot_General.Command.ClampB_Open;
				_DO6.ByPassClampSensor := GVL_ADS.FanucRobot_General.Command.ByPassClampSensor;
				GVL_ADS.FanucRobot_General.Status.ClampA_Open := _DI1.ClampA_Open;
				GVL_ADS.FanucRobot_General.Status.ClampA_Sensor := _DI1.ClampA_Sensor;
				GVL_ADS.FanucRobot_General.Status.ClampB_Open := _DI1.ClampB_Open ;
				GVL_ADS.FanucRobot_General.Status.ClampB_Sensor := _DI1.ClampB_Sensor;
				_VelocityCommand.nInt := GVL_ADS.FanucRobot_General.Command.RobotVelocity;
        END_CASE

        IF (*qFault OR *)_Error THEN
            //Soft E-Stop will cause Fault error
            eState := E_MethodStatus_Basic.STATE_ERROR;
        ELSIF _Abort THEN
            eState := E_MethodStatus_Basic.STATE_ABORTING;
		ELSIF Estop THEN
			eState := E_MethodStatus_Basic.STATE_ABORTING;
        END_IF
    E_MethodStatus_Basic.STATE_DONE:
        ;
    E_MethodStatus_Basic.STATE_ABORTING:
	;
//        Hold();

        IF _UO1.UO04_PrgPaused THEN
            eState := E_MethodStatus_Basic.STATE_Aborted;
        END_IF
    E_MethodStatus_Basic.STATE_Aborted:
        IF _UI1.UI05_FaultReset OR GVL.Reset THEN
            eState := E_MethodStatus_Basic.STATE_RESETTING;
        END_IF
    E_MethodStatus_Basic.STATE_ERROR:
        IF _UI1.UI05_FaultReset THEN
            eState := E_MethodStatus_Basic.STATE_RESETTING;
        END_IF
    E_MethodStatus_Basic.STATE_RESETTING:
        CASE uiRobotResettingStep OF
            0:
                IF NOT _UO1.UO06_Fault THEN
                    IF NOT _UO1.UO04_PrgPaused THEN
                        uiRobotResettingStep := 1000;
                    ELSE
                        uiRobotResettingStep := 2000;
                    END_IF
                ELSE
                    uiRobotResettingStep := 1000;
                END_IF
            1000:
                M_Reset(TRUE);
				TON_Reset_delay.in := TRUE;
				IF TON_Reset_delay.Q THEN
                	uiRobotResettingStep := 1010;
				END_IF
            1010:
				TON_Reset_delay.IN :=FALSE;
                M_Reset(FALSE);
                uiRobotResettingStep := 9000;
            2000:
                _UI1.UI02_Hold       := TRUE;
                TON_Restart_delay.IN := TRUE; // TimeCount start

                IF TON_Restart_delay.Q THEN
                    uiRobotResettingStep := 2100;
                END_IF
            2100:
                TON_Restart_delay.IN := FALSE;
                _UI1.UI06_Start      := TRUE;
                uiRobotResettingStep := 9000;
            9000:
                IF NOT qFault THEN
                    eState := E_MethodStatus_Basic.STATE_DORMANT;
                END_IF
        END_CASE
END_CASE
Rtrig_RebootRobot(CLK:= GVL.MachineReset.AllReset);
IF Rtrig_RebootRobot.Q	AND qFault THEN
	ReBoot();
END_IF
END_ACTION

PROPERTY AbsMoveClampA_Handshake : ST_Fanuc_AbsMove
GET
AbsMoveClampA_Handshake := _DO3;
END_GET
SET
// Outside -> FB 
_DO3 := AbsMoveClampA_Handshake;
END_SET
END_PROPERTY

PROPERTY AbsMoveClampB_Handshake : ST_Fanuc_AbsMove
GET
AbsMoveClampB_Handshake := _DO4;
END_GET
SET
// Outside -> FB 
_DO4 := AbsMoveClampB_Handshake;
END_SET
END_PROPERTY

PROPERTY Bzone_AllowWork : Bool
GET
Bzone_AllowWork := THIS^._DO6.Bzone_AllowWork;
END_GET
SET
 THIS^._DO6.Bzone_AllowWork :=Bzone_AllowWork ;
END_SET
END_PROPERTY

PROPERTY BZoneInWork : Bool
GET
BZoneInWork := THIS^._DI12.BzoneInWork;
END_GET
END_PROPERTY

PROPERTY Command : ST_FanucUO1
GET
Command := _UO1;
END_GET
SET
_UO1 := Command;
END_SET
END_PROPERTY

METHOD Enable : BOOL
VAR_INPUT
iTrigger:BOOL;
END_VAR
VAR
	_RobotEnable:BOOL;
END_VAR
_RobotEnable:=iTrigger (*AND NOT Fault()*);

_UI1.UI01_IMSP:=_RobotEnable;
_UI1.UI02_Hold:=_RobotEnable;
_UI1.UI03_SFSP:=_RobotEnable;
_UI1.UI08_Enable:=_RobotEnable;
END_METHOD

METHOD EStop
VAR_INPUT
END_VAR
_UI1.UI03_SFSP:=FALSE;
END_METHOD

PROPERTY FanucRobot_MotionStatus : ST_Fanuc_Status
GET
FanucRobot_MotionStatus := _DI1;
END_GET
END_PROPERTY

METHOD Fault : BOOL
VAR_INPUT
END_VAR
VAR_INST
	bConectionError : BOOL;
END_VAR
bConectionError := (_EIPConnectionState <>0) OR (_FanucEIPState <> 0);
Fault:=_UO1.UO06_Fault OR _UO1.UO09_BattAlarm OR _DI1.Error OR bConectionError OR _UO1.UO08_TPEnabled;
END_METHOD

METHOD GetModelState
VAR_INPUT
END_VAR
VAR_OUTPUT
    xDone : BOOL;
    xBusy : BOOL;
    xError : BOOL;
    xAborted : BOOL;
    iErrorID : UDINT;
	UniqueErrorCode : STRING;
END_VAR
xError := Error;
iErrorID := INT_TO_UDINT(ErrorCode.nInt);
END_METHOD

METHOD GetName : STRING
VAR_INPUT
END_VAR
GetName := 'Fanuc Robot';
END_METHOD

METHOD Hold
VAR_INPUT
END_VAR
_UI1.UI02_Hold:=FALSE;
END_METHOD

PROPERTY Homed : Bool
GET
Homed := _RSR2_Completed OR _UO1.UO07_AtPerch;
END_GET
END_PROPERTY

PROPERTY LayerIndex : INT
SET
_Do15 := LayerIndex;
END_SET
END_PROPERTY

METHOD M_ActiveRSR01
VAR_INPUT
END_VAR
VAR_OUTPUT
	bCompleted : BOOL;
END_VAR
CASE eState OF
    E_MethodStatus_Basic.STATE_DORMANT:
        Enable(FALSE);
        M_Reset(FALSE);
        _uiRSR01_Step        := 0;
        uiRobotExecutingStep := 0;
        uiRobotResettingStep := 0;
        _RSR1_Ready          := FALSE;
        _RSR2_Completed      := FALSE;
        _RSR3_Ready          := FALSE;
        TON_Reset_delay.IN   := FALSE;
        _RSR1_Ready          := FALSE;

        IF _eOpMode = RSR01 OR _eOpMode = RSR02 OR _eOpMode = RSR03 THEN
            eState := E_MethodStatus_Basic.STATE_EXECUTING;
        END_IF
    E_MethodStatus_Basic.STATE_EXECUTING:
        CASE uiRobotExecutingStep OF
            0:
                Enable(iTrigger := TRUE);
                TON_Restart_delay.IN := TRUE;

                IF TON_Restart_delay.Q THEN
                    uiRobotExecutingStep := 10;
                END_IF
            10:
                TON_Restart_delay.IN := FALSE;
                M_Reset(iTrigger := TRUE);
                _UI1.UI04_CycleStop  := TRUE;
                TON_ResetFixDelay.IN := TRUE;

                IF TON_ResetFixDelay.Q THEN
                    uiRobotExecutingStep := 100;
                END_IF
            100:
                TON_ResetFixDelay.IN := FALSE;
                TON_Reset_delay.in   := TRUE;
                M_Reset(iTrigger := FALSE);
                _UI1.UI04_CycleStop := FALSE;

                IF TON_Reset_delay.Q THEN
                    IF _UO1.UO01_CmdEnabled AND _UO1.UO02_SystemReady THEN
                        _Error                := FALSE;
						Enable(iTrigger := TRUE); // 20250428 Albert
                        _VelocityCommand.nInt := 1;
                        uiRobotExecutingStep  := 200;
                    ELSIF Error THEN
                        eState := E_MethodStatus_Basic.STATE_ERROR;
                    END_IF
                END_IF
            200:
                // Clear Fanuc robot's action
                TON_Reset_delay.IN                                            := FALSE;
                GVL_ADS.AutoMode_WarehouseMotoWithRobotMove.HandShake.Execute := FALSE;
                GVL_ADS.AutoMode_RobotAbsMove.HandShake.Execute               := FALSE;
                _DO1.bExecute                                                 := FALSE; // Warehouse with robot clampA
                _DO2.bExecute                                                 := FALSE; // Warehouse with robot clampB
                _DO3.bExecute                                                 := FALSE; // AbsMove with robot clampA
                _DO4.bExecute                                                 := FALSE; // AbsMove with robot clampB
                uiRobotExecutingStep                                          := 300;
            300:
                // Active RSR1
                _UI1.UI09_RSR1         := TRUE;
                Ton_SetProgTimeOut.IN  := TRUE; // Switch to RSR1 start.
                Ton_RSR_SwitchDelay.IN := TRUE;

                IF _UO1.UO11_ACK1 THEN
                    uiRobotExecutingStep := 400;
                ELSIF Error OR Ton_SetProgTimeOut.Q THEN
                    _Error  := TRUE;
                    _Status := 'RSR1 has error when RSR1 active.';
                END_IF
            400:
                // Close RSR1 command
                Ton_SetProgTimeOut.IN := FALSE; // Switch to RSR1 close.

                IF Ton_RSR_SwitchDelay.Q THEN
                    _UI1.UI09_RSR1       := FALSE;
                    uiRobotExecutingStep := 500;
                END_IF
            500:
                // Allow Robot auto / manual job
                IF (GVL_ADS.AutoMode_RobotAbsMove.HandShake.Busy OR GVL_ADS.AutoMode_RobotAbsMove.HandShake.Done) AND
                    (GVL_ADS.AutoMode_WarehouseMotoWithRobotMove.HandShake.Busy OR GVL_ADS.AutoMode_WarehouseMotoWithRobotMove.HandShake.Done) (*AND
                    (GVL_ADS.ADS_MotoCalibrationData.WDataCore.HandShake.Busy OR GVL_ADS.ADS_MotoCalibrationData.WDataCore.HandShake.Done) AND
                    (GVL_ADS.ADS_MotoCalibrationData.AbslutCore.HandShake.Busy OR GVL_ADS.ADS_MotoCalibrationData.AbslutCore.HandShake.Done)*)
                    THEN
                    bCompleted := FALSE;
                ELSE
                    bCompleted := TRUE;
                END_IF
				M_ManualService();
                //_VelocityCommand.nInt                           := GVL_ADS.FanucRobot_General.Command.RobotVelocity;
                _RSR1_Ready                                     := TRUE;

                IF _DI1.Error THEN
                    _Abort := TRUE;
                END_IF
        END_CASE

        IF _Abort THEN
            eState := E_MethodStatus_Basic.STATE_ABORTING;
        ELSIF Hold THEN
            eState := E_MethodStatus_Basic.STATE_Holding;
		ELSIF _UO1.UO06_Fault THEN
	        //_Abort := TRUE;

//			_Error  := TRUE;
//			_Status := 'Robot has fatal alarm';
//			eState  := E_MethodStatus_Basic.STATE_ERROR;
        END_IF
    E_MethodStatus_Basic.STATE_DONE:
        ;
    E_MethodStatus_Basic.STATE_ABORTING:
        eState := E_MethodStatus_Basic.STATE_ERROR;
    E_MethodStatus_Basic.STATE_Aborted:
        ;
    E_MethodStatus_Basic.STATE_ERROR:
        Enable(iTrigger := FALSE);
        _RSR1_Ready := FALSE;

        IF reset THEN
            eState := E_MethodStatus_Basic.STATE_RESETTING;
        END_IF

        IF NOT Estop AND NOT Error THEN
            eState := E_MethodStatus_Basic.STATE_RESETTING;
        END_IF
    E_MethodStatus_Basic.STATE_RESETTING:
		CASE uiRobotResettingStep OF
			0 : 
				_Error                   := FALSE;
				_Abort := false;
				_Status                  := '';
				M_ResetAllCommand();
				Ton_START_SwitchDelay.IN := FALSE;
				TON_Restart_delay.IN := FALSE;
				uiRobotResettingStep := 10;
			10:
				M_Reset(iTrigger :=TRUE);
				TON_Restart_delay.IN := TRUE;
				IF TON_Restart_delay.Q THEN
					M_EnableWith4Input(TRUE	,TRUE,TRUE,FALSE);
					uiRobotResettingStep := 20;
				END_IF
			20:
				TON_Restart_delay.IN := FALSE;
				M_Reset(iTrigger :=FALSE);
        		//Enable(iTrigger := TRUE);
				IF NOT  _UO1.UO06_Fault THEN
					M_EnableWith4Input(TRUE	,TRUE,TRUE,FALSE);
					uiRobotResettingStep := 50;
				END_IF
				IF reset THEN
					uiRobotResettingStep := 0;
				END_IF
			30 :
				M_Reset(iTrigger :=TRUE);
				uiRobotResettingStep := 40;
			40:
				M_Reset(iTrigger :=FALSE);
				uiRobotResettingStep := 50;
			50:
				IF reset THEN
					uiRobotResettingStep := 0;
				END_IF
				IF NOT Error THEN
					eState := E_MethodStatus_Basic.STATE_DORMANT;
				END_IF
		END_CASE
    E_MethodStatus_Basic.STATE_Holding:
        _UI1.UI02_Hold := FALSE;

        IF _UO1.UO04_PrgPaused AND NOT _UO1.UO03_PrgRunning THEN
            Halt    := TRUE;
            _Status := 'Robot in Halt State';
            eState  := E_MethodStatus_Basic.STATE_Held;
        END_IF
		IF reset THEN
			eState         := E_MethodStatus_Basic.STATE_ERROR;
		END_IF
    E_MethodStatus_Basic.STATE_Held:
		Ton_START_SwitchDelay.IN := FALSE;
        IF reset AND NOT Hold THEN
			//M_Reset(iTrigger:=TRUE);		//edit by min , if need resume robot motion dont set robot UI04 cyclestop
			_UI1.UI05_FaultReset:=TRUE;
            Halt := FALSE;
		ELSE
			M_Reset(iTrigger :=FALSE);
        END_IF

        IF NOT Halt AND Start THEN
            _UI1.UI02_Hold := TRUE;
            eState         := E_MethodStatus_Basic.STATE_UnHold;
        END_IF
    E_MethodStatus_Basic.STATE_UnHold:
        Ton_START_SwitchDelay.IN := TRUE;
		 _UI1.UI09_RSR1         := TRUE;
        _UI1.UI06_Start          := NOT Ton_START_SwitchDelay.Q;
		
        IF NOT _UO1.UO04_PrgPaused AND _UO1.UO03_PrgRunning AND NOT _UI1.UI06_Start THEN
            Ton_START_SwitchDelay.IN := FALSE;
			 _UI1.UI09_RSR1         := FALSE;
            eState                   := E_MethodStatus_Basic.STATE_EXECUTING;
        END_IF
END_CASE

IF Estop THEN
   // _Error  := TRUE;
    _Status := 'EStop has been trigged.';
	eState  := E_MethodStatus_Basic.STATE_ERROR;
ELSIF _UO1.UO08_TPEnabled THEN
    _Error  := TRUE;
    _Status := 'TP has got contol';
	eState  := E_MethodStatus_Basic.STATE_ERROR;
ELSIF _UO1.UO09_BattAlarm THEN
    _Error  := TRUE;
    _Status := 'Robot has Battary alarm';
	eState  := E_MethodStatus_Basic.STATE_ERROR;
END_IF
END_METHOD

METHOD M_ActiveRSR02
VAR_INPUT
END_VAR
VAR_OUTPUT
	bCompleted : BOOL;
END_VAR
CASE eState OF
	E_MethodStatus_Basic.STATE_DORMANT:
        Enable(FALSE);
        M_Reset(FALSE);
        _uiRSR01_Step := 0;
		uiRobotExecutingStep := 0;
        uiRobotResettingStep := 0;
		_RSR1_Ready := FALSE;
		_RSR2_Completed := FALSE;
		_RSR3_Ready:=FALSE;
		TON_Reset_delay.IN := FALSE;
		IF _eOpMode = RSR01 OR _eOpMode = RSR02 OR _eOpMode = RSR03 THEN
			eState := E_MethodStatus_Basic.STATE_EXECUTING;
		END_IF
	E_MethodStatus_Basic.STATE_EXECUTING:
		CASE uiRobotExecutingStep OF
			0:
                Enable(iTrigger := TRUE);
				TON_Restart_delay.IN := TRUE;
				IF TON_Restart_delay.Q THEN
					uiRobotExecutingStep := 10;
				END_IF
			10:
				TON_Restart_delay.IN := FALSE;
                M_Reset(iTrigger := TRUE);
				TON_ResetFixDelay.in := TRUE;
				_UI1.UI04_CycleStop := TRUE;
				IF TON_ResetFixDelay.Q THEN
	                uiRobotExecutingStep := 100;
				END_IF
			100:
				TON_ResetFixDelay.in := FALSE;
				TON_Reset_delay.in := TRUE;
                M_Reset(iTrigger := FALSE);
				_UI1.UI04_CycleStop := FALSE;
				IF TON_Reset_delay.Q THEN
					IF _UO1.UO01_CmdEnabled AND _UO1.UO02_SystemReady THEN
						_VelocityCommand.nInt := 1;
						uiRobotExecutingStep := 200;
					ELSIF Error THEN
						eState := E_MethodStatus_Basic.STATE_ERROR;
					END_IF
				END_IF
			200:
				// Clear Fanuc robot's action
				GVL_ADS.AutoMode_WarehouseMotoWithRobotMove.HandShake.Execute := FALSE;
				GVL_ADS.AutoMode_RobotAbsMove.HandShake.Execute := FALSE;
				_DO1.bExecute := FALSE;
				_DO2.bExecute := FALSE;
				_DO3.bExecute := FALSE;
				_DO4.bExecute := FALSE;
				uiRobotExecutingStep := 300;
			300:
				// Switch RSR02
				_UI1.UI10_RSR2 := TRUE;
		
				IF _UO1.UO12_ACK2 THEN
					uiRobotExecutingStep := 400;
				END_IF
			400:
				_UI1.UI10_RSR2 := FALSE;
				IF (_DI1.Done OR _UO1.UO07_AtPerch )  
				THEN
					uiRobotExecutingStep := 9900;
				END_IF
			9900:
				eState := E_MethodStatus_Basic.STATE_DONE;
		END_CASE
	E_MethodStatus_Basic.STATE_DONE:
		_RSR2_Completed := TRUE;
		bCompleted := TRUE;
	E_MethodStatus_Basic.STATE_ABORTING:
		;
	E_MethodStatus_Basic.STATE_Aborted:
		;
	E_MethodStatus_Basic.STATE_ERROR:
		Enable(iTrigger := FALSE);
		IF reset THEN
			eState := E_MethodStatus_Basic.STATE_RESETTING;
		END_IF
		IF NOT Estop AND NOT Error THEN
			eState := E_MethodStatus_Basic.STATE_RESETTING;
		END_IF
	E_MethodStatus_Basic.STATE_RESETTING:
		eState := E_MethodStatus_Basic.STATE_DORMANT;
END_CASE
IF Estop OR _UO1.UO08_TPEnabled THEN
	eState := E_MethodStatus_Basic.STATE_ERROR;
	_Error := TRUE;
	_Status := 'EStop has been trigged.';
END_IF
END_METHOD

METHOD M_ActiveRSR03
VAR_INPUT
END_VAR
VAR_OUTPUT
	bCompleted : BOOL;
END_VAR
CASE _uiRSR03_Step OF
	0:
		// Stop Prog
		_RSR1_Ready := FALSE;
		_RSR2_Completed := FALSE;
		_RSR3_Ready:=FALSE;
		_UI1.UI04_CycleStop := TRUE;
		IF NOT _UO1.UO04_PrgPaused AND NOT _UO1.UO03_PrgRunning THEN
			_uiRSR03_Step := 100;
		END_IF
	100:
		// Close cycle stop
		_UI1.UI04_CycleStop := FALSE;
		// Set current prog - RSR03
		_UI1.UI11_RSR3 := TRUE;
		IF _UO1.UO13_ACK3 THEN
			_uiRSR03_Step := 200;
		END_IF
	200:
		// Clear RSR03 command 
		_UI1.UI11_RSR3 := FALSE;
		_uiRSR03_Step := 300;
	300:
		// Allow Read / Write offset data
		IF ( GVL_ADS.FanucRobot_ReadAllOffsetData.Status.Busy  OR GVL_ADS.FanucRobot_ReadAllOffsetData.Status.Done) AND
			(GVL_ADS.FanucRobot_ReadSingleOffsetData.Status.Busy OR GVL_ADS.FanucRobot_ReadSingleOffsetData.Status.Done) AND
			(GVL_ADS.FanucRobot_WirteSingleOffsetData.Status.Busy OR GVL_ADS.FanucRobot_WirteSingleOffsetData.Status.Done ) AND
			(GVL_ADS.FanucRobot_WriteAllOffsetData.Status.Busy OR GVL_ADS.FanucRobot_WriteAllOffsetData.Status.Done) 
		THEN
			_RSR3_Ready := FALSE;
			bCompleted := FALSE;
		ELSE
			_RSR3_Ready := FALSE;
			bCompleted := TRUE;
		END_IF 
		
END_CASE

CASE eState OF
	E_MethodStatus_Basic.STATE_DORMANT:
        Enable(FALSE);
        M_Reset(FALSE);
        _uiRSR01_Step := 0;
		uiRobotExecutingStep := 0;
        uiRobotResettingStep := 0;
		_RSR1_Ready := FALSE;
		_RSR2_Completed := FALSE;
		_RSR3_Ready:=FALSE;
		TON_Reset_delay.IN := FALSE;
		IF _eOpMode = RSR01 OR _eOpMode = RSR02 OR _eOpMode = RSR03 THEN
			eState := E_MethodStatus_Basic.STATE_EXECUTING;
		END_IF
	E_MethodStatus_Basic.STATE_EXECUTING:
		CASE uiRobotExecutingStep OF
			0:
                Enable(iTrigger := TRUE);
				TON_Restart_delay.IN := TRUE;
				IF TON_Restart_delay.Q THEN
					uiRobotExecutingStep := 10;
				END_IF
			10:
				TON_Restart_delay.IN := FALSE;
                M_Reset(iTrigger := TRUE);
				_UI1.UI04_CycleStop := TRUE;
				TON_ResetFixDelay.IN := TRUE;
				IF TON_ResetFixDelay.Q THEN
                	uiRobotExecutingStep := 100;
				END_IF
			100:
				TON_ResetFixDelay.IN := FALSE;
				TON_Reset_delay.in := TRUE;
                M_Reset(iTrigger := FALSE);
				_UI1.UI04_CycleStop := FALSE;
				IF TON_Reset_delay.Q THEN
					IF _UO1.UO01_CmdEnabled AND _UO1.UO02_SystemReady THEN
						_VelocityCommand.nInt := 1;
						uiRobotExecutingStep := 200;
					ELSIF Error THEN
						eState := E_MethodStatus_Basic.STATE_ERROR;
					END_IF
				END_IF
			200:
				// Clear Fanuc robot's action
				TON_Reset_delay.IN := FALSE;
				GVL_ADS.AutoMode_WarehouseMotoWithRobotMove.HandShake.Execute := FALSE;
				GVL_ADS.AutoMode_RobotAbsMove.HandShake.Execute := FALSE;
				_DO1.bExecute := FALSE; // Warehouse with robot clampA
				_DO2.bExecute := FALSE; // Warehouse with robot clampB
				_DO3.bExecute := FALSE; // AbsMove with robot clampA
				_DO4.bExecute := FALSE; // AbsMove with robot clampB
				uiRobotExecutingStep := 300;
			300:
				// Active RSR1
                _UI1.UI11_RSR3 := TRUE;
                IF _UO1.UO13_ACK3 THEN
                    uiRobotExecutingStep := 400;
				ELSIF Error THEN
					_Error := TRUE;
					_Status:='RSR3 has error when RSR3 active.';
                END_IF
			400:
				// Allow Read / Write offset data
				IF ( GVL_ADS.FanucRobot_ReadAllOffsetData.Status.Busy  OR GVL_ADS.FanucRobot_ReadAllOffsetData.Status.Done) AND
					(GVL_ADS.FanucRobot_ReadSingleOffsetData.Status.Busy OR GVL_ADS.FanucRobot_ReadSingleOffsetData.Status.Done) AND
					(GVL_ADS.FanucRobot_WirteSingleOffsetData.Status.Busy OR GVL_ADS.FanucRobot_WirteSingleOffsetData.Status.Done ) AND
					(GVL_ADS.FanucRobot_WriteAllOffsetData.Status.Busy OR GVL_ADS.FanucRobot_WriteAllOffsetData.Status.Done) 
				THEN
					_RSR3_Ready := FALSE;
					bCompleted := FALSE;
				ELSE
					_RSR3_Ready := FALSE;
					bCompleted := TRUE;
				END_IF 
		END_CASE
	E_MethodStatus_Basic.STATE_DONE:
		;
	E_MethodStatus_Basic.STATE_ABORTING:
		;
	E_MethodStatus_Basic.STATE_Aborted:
		;
	E_MethodStatus_Basic.STATE_ERROR:
		Enable(iTrigger := FALSE);
		IF Reset THEN
			eState := E_MethodStatus_Basic.STATE_RESETTING;
		END_IF
		IF  Estop AND NOT Error THEN
			eState := E_MethodStatus_Basic.STATE_RESETTING;
		END_IF
	E_MethodStatus_Basic.STATE_RESETTING:
		eState := E_MethodStatus_Basic.STATE_DORMANT;
END_CASE

IF Estop OR _UO1.UO08_TPEnabled THEN
	eState := E_MethodStatus_Basic.STATE_ERROR;
	_Error := TRUE;
	_Status := 'EStop has been trigged.';
END_IF
END_METHOD

METHOD M_ClearState : BOOL;
VAR_INPUT
END_VAR

eState := E_MethodStatus_Basic.STATE_DORMANT;
uiRobotExecutingStep := 0;
uiRobotResettingStep := 0;
M_ClearState := TRUE;
END_METHOD

METHOD M_ControlRSR01
VAR_INPUT
END_VAR
VAR_OUTPUT
	bCompleted : BOOL;
	ModeChanging : BOOL;
	ModeChanged : BOOL;
END_VAR
ModeChanging := FALSE;
ModeChanged := TRUE;
M_ActiveRSR01(bCompleted => bCompleted);

IF OpMode <> _eOpMode AND bCompleted THEN
    _uiRSR01_Step := 0;
    eState := E_MethodStatus_Basic.STATE_DORMANT;
    _eOpMode := OpMode;
END_IF
END_METHOD

METHOD M_ControlRSR02
VAR_INPUT
END_VAR
VAR_OUTPUT
    bCompleted : BOOL;
    ModeChanging : BOOL;
    ModeChanged : BOOL;
END_VAR
ModeChanging := FALSE;
ModeChanged := TRUE;
M_ActiveRSR02(bCompleted => bCompleted);

IF OpMode <> _eOpMode AND bCompleted THEN
    _uiRSR02_Step := 0;
    eState := E_MethodStatus_Basic.STATE_DORMANT;
    _eOpMode := OpMode;
END_IF
END_METHOD

METHOD M_ControlRSR03

VAR_INPUT
END_VAR
VAR_OUTPUT
    bCompleted : BOOL;
    ModeChanging : BOOL;
    ModeChanged : BOOL;
END_VAR
ModeChanging := FALSE;
ModeChanged := TRUE;
M_ActiveRSR03(bCompleted => bCompleted);

IF OpMode <> _eOpMode AND bCompleted THEN
	_uiRSR03_Step := 0;
	eState := E_MethodStatus_Basic.STATE_DORMANT;
	_eOpMode := OpMode;
END_IF
END_METHOD

METHOD PRIVATE M_EnableWith4Input : BOOL
VAR_INPUT
	IMSP : BOOL;
	Hold : BOOL;
	SFSP : BOOL;
	Enable : BOOL;
END_VAR
_UI1.UI01_IMSP:=IMSP;
_UI1.UI02_Hold:=Hold;
_UI1.UI03_SFSP:=SFSP;
_UI1.UI08_Enable:=Enable;
END_METHOD

METHOD M_GetErrorCode : Int
VAR_INPUT
END_VAR
ErrorCode.BitList.Bit0 := _DI1.ErrorID_01;
ErrorCode.BitList.Bit1 := _DI1.ErrorID_02;
ErrorCode.BitList.Bit2 := _DI1.ErrorID_03;
ErrorCode.BitList.Bit3 := _DI1.ErrorID_04;
ErrorCode.BitList.Bit4 := _DI1.ErrorID_05;
ErrorCode.BitList.Bit5 := _DI1.ErrorID_06;
ErrorCode.BitList.Bit6 := _DI1.ErrorID_07;
ErrorCode.BitList.Bit7 := _DI1.ErrorID_08;
//ErrorCode.BitList.Bit8 := _DI1.ErrorID_09;
//ErrorCode.BitList.Bit9 := _DI1.ErrorID_10;
M_GetErrorCode := ErrorCode.nInt;
END_METHOD

METHOD M_Kawasaki_API
VAR_INPUT
	WarehouseClampA_Handshake : UINT;
	WarehouseClampB_Handshake : UINT;
	AbsMoveClampA_Handshake : UINT;
	AbsMoveClampB_Handshake : UINT;
END_VAR
VAR_OUTPUT
	Status : UINT;
END_VAR
MEMMOVE(destAddr:=ADR(_DO1),srcAddr:=ADR(WarehouseClampA_Handshake),n:=2);
MEMMOVE(destAddr:=ADR(_DO2),srcAddr:=ADR(WarehouseClampB_Handshake),n:=2);
MEMMOVE(destAddr:=ADR(_DO3),srcAddr:=ADR(AbsMoveClampA_Handshake),n:=2);
MEMMOVE(destAddr:=ADR(_DO4),srcAddr:=ADR(AbsMoveClampB_Handshake),n:=2);
IF NOT _UO1.UO08_TPEnabled THEN
	MEMMOVE(destAddr:=ADR(Status),srcAddr:=ADR(_DI1),n:=2);
END_IF
END_METHOD

METHOD M_ManualService
VAR_INPUT
END_VAR
_DO5.ClampA_Close := ManualCtrl.ClampA_Close;
_DO5.ClampA_Open := ManualCtrl.ClampA_Open;
_DO5.ClampB_Close := ManualCtrl.ClampB_Close;
_DO5.ClampB_Open := ManualCtrl.ClampB_Open;
_DO6.ByPassClampSensor := ManualCtrl.ByPassClampSensor;
GVL_ADS.FanucRobot_General.Status.ClampA_Open := _DI1.ClampA_Open;
GVL_ADS.FanucRobot_General.Status.ClampA_Sensor := _DI1.ClampA_Sensor;
GVL_ADS.FanucRobot_General.Status.ClampB_Open := _DI1.ClampB_Open;
GVL_ADS.FanucRobot_General.Status.ClampB_Sensor := _DI1.ClampB_Sensor;
END_METHOD

METHOD M_Reset : BOOL
VAR_INPUT
	iTrigger:BOOL;
END_VAR
_UI1.UI05_FaultReset:=iTrigger;
_UI1.UI04_CycleStop:=iTrigger;
END_METHOD

METHOD M_ResetAbsMoveClampACommand : BOOL
VAR_INPUT
END_VAR
VAR
	SpareData : ST_Fanuc_AbsMove;
END_VAR
_DO3 := SpareData;

M_ResetAbsMoveClampACommand := TRUE; // Method end
END_METHOD

METHOD M_ResetAbsMoveClampBCommand : BOOL
VAR_INPUT
END_VAR
VAR
	SpareData : ST_Fanuc_AbsMove;
END_VAR
_DO4 := SpareData;

M_ResetAbsMoveClampBCommand := true; // Method end
END_METHOD

METHOD M_ResetAbsMoveCommand : BOOL
VAR_INPUT
END_VAR
// Clear AbsMove ClampA command data
M_ResetAbsMoveClampACommand();
// Clear AbsMove ClampB command data
M_ResetAbsMoveClampBCommand();

M_ResetAbsMoveCommand := TRUE; // Method end
END_METHOD

METHOD M_ResetAllCommand : BOOL
VAR_INPUT
END_VAR
// Clear WareHouse command
M_ResetWareHouseCommand();
// Clear AbsMove Command
M_ResetAbsMoveCommand();

M_ResetAllCommand := TRUE; // Method end
END_METHOD

METHOD M_ResetMoveBoxToFeedInConveyor_ClampA : BOOL
VAR_INPUT
END_VAR
VAR
	SpaceData : ST_Fanuc_AbsMove;
END_VAR
_DO3 := SpaceData;

M_ResetMoveBoxToFeedInConveyor_ClampA := TRUE; // Mehtod end
END_METHOD

METHOD M_ResetMoveBoxToFeedInConveyor_ClampB : BOOL
VAR_INPUT
END_VAR
VAR
    SpaceData : ST_Fanuc_AbsMove;
END_VAR
_DO4 := SpaceData;

M_ResetMoveBoxToFeedInConveyor_ClampB := TRUE; // Method end
END_METHOD

METHOD M_ResetMoveBoxToFeedInConveyor_ClampBoth : BOOL
VAR_INPUT
END_VAR
VAR
    SpaceData : ST_Fanuc_AbsMove;
END_VAR
_DO3 := SpaceData;
_DO4 := SpaceData;

M_ResetMoveBoxToFeedInConveyor_ClampBoth := TRUE; // Method end
END_METHOD

METHOD M_ResetMoveBoxToRoundBelt_Both : BOOL
VAR_INPUT
END_VAR
VAR
    SpaceData : ST_Fanuc_AbsMove;
END_VAR
_DO3 := SpaceData;
_DO4 := SpaceData;

M_ResetMoveBoxToRoundBelt_Both := TRUE; // Method end
END_METHOD

METHOD M_ResetPullOutConveyorPickUpBox_ClampA : BOOL
VAR_INPUT
END_VAR
VAR
	SpaceData : ST_Fanuc_AbsMove;
END_VAR
_DO3 := SpaceData;

M_ResetPullOutConveyorPickUpBox_ClampA := TRUE; // Method end
END_METHOD

METHOD M_ResetPullOutConveyorPickUpBox_ClampB : BOOL
VAR_INPUT
END_VAR
VAR
    SpaceData : ST_Fanuc_AbsMove;
END_VAR
_DO4 := SpaceData;

M_ResetPullOutConveyorPickUpBox_ClampB := true; // Method end
END_METHOD

METHOD M_ResetPullOutConveyorPickUpBox_ClampBoth : BOOL
VAR_INPUT
END_VAR
VAR
    SpaceData : ST_Fanuc_AbsMove;
END_VAR
_DO3 := SpaceData;
_DO4 := SpaceData;

M_ResetPullOutConveyorPickUpBox_ClampBoth := TRUE; // Method end
END_METHOD

METHOD PUBLIC M_ResetRobotAbsMove : BOOL
VAR_INPUT
	ResetClampA : BOOL;
	ResetClampB : BOOL;
END_VAR

VAR
	SpaceData : ST_Fanuc_AbsMove;
END_VAR
IF ResetClampA THEN
	_DO3 := SpaceData;
END_IF

IF ResetClampB THEN
	_DO4 := SpaceData;
END_IF

M_ResetRobotAbsMove:=True;
END_METHOD

METHOD M_ResetWareHouseClampACommand : BOOL
VAR_INPUT
END_VAR
VAR
	SpareData : ST_Fanuc_WarehouseHandshake;
END_VAR
_DO1 := SpareData;

M_ResetWareHouseClampACommand := TRUE; // Method end
END_METHOD

METHOD M_ResetWareHouseClampBCommand : BOOL
VAR_INPUT
END_VAR
VAR
	SpareData : ST_Fanuc_WarehouseHandshake;
END_VAR
_DO2 := SpareData;

M_ResetWareHouseClampBCommand := true; // Method end
END_METHOD

METHOD M_ResetWareHouseCommand : BOOL
VAR_INPUT
END_VAR
// Clear WareHouse ClampA command data
M_ResetWareHouseClampACommand();
// Clear WareHouse ClampB command data
M_ResetWareHouseClampBCommand();

M_ResetWareHouseCommand := TRUE; // Method end
END_METHOD

METHOD M_ResetWareHousePickUpBox_ClampA : BOOL
VAR_INPUT
END_VAR
VAR
	SpaceData :ST_Fanuc_WarehouseHandshake;
END_VAR
// Clear command
_DO1 := SpaceData;

M_ResetWareHousePickUpBox_ClampA := TRUE; // Method End
END_METHOD

METHOD M_ResetWareHousePickUpBox_ClampB : BOOL
VAR_INPUT
END_VAR
VAR
	SpaceData :ST_Fanuc_WarehouseHandshake;
END_VAR
// Clear command
_DO2 := SpaceData;

M_ResetWareHousePickUpBox_ClampB := TRUE; // Method End
END_METHOD

METHOD M_ResetWareHousePickUpBox_ClampBoth : BOOL
VAR_INPUT
END_VAR
VAR
	SpaceData :ST_Fanuc_WarehouseHandshake;
END_VAR
// Clear command
_DO1 := SpaceData;
_DO2 := SpaceData;

M_ResetWareHousePickUpBox_ClampBoth := TRUE; // Method end
END_METHOD

(* This Method is used to send command data to Fanuc Robot, only clampA is work 
*)
METHOD M_StartAbsMoveAction_ClampA : BOOL
VAR_INPUT
	TargetArea : E_RobotArea; // Select the zone where robot will going.
	TargetAddress : E_RobotAddress; // Because the address num in different zone, the number define is different. But also need >= 1, 0 = undefined
	ClampAction : E_ClampAction; // need to define the command
	BoxReady : BOOL; // Fanuc robot prog will stop at a safe position just before reaching the target location, until `AllowContinue` is set to true.
END_VAR

VAR_OUTPUT
    Error  : BOOL;
    ErrMsg : T_MaxString;
END_VAR

VAR_INST
	_Area : ST_IntToBool;
	_Address : ST_IntToBool;
END_VAR
// Set target area
_Area.nInt := TargetArea;

CASE TargetArea OF
    E_RobotArea.RoundBelt..E_RobotArea.PullOutConveyor:
        _Area.nInt := TargetArea;
ELSE
    Error  := TRUE;
    ErrMsg := 'ClampA target area out of range';
	RETURN;
END_CASE

// Set target address
_Address.nInt := TargetAddress;

CASE TargetAddress OF
    E_RobotAddress.Address01..E_RobotAddress.Address06:
        _Address.nInt := TargetAddress;
ELSE
    Error  := TRUE;
    ErrMsg := 'ClampA target address out of range';
	RETURN;
END_CASE

// Check ClampA Action is correct
CASE ClampAction OF
	E_ClampAction.PickUp:
		_DO3.bGet := TRUE;
	E_ClampAction.Place:
		_DO3.bGet := FALSE;
ELSE
	Error := TRUE;
	ErrMsg := 'ClampA Action is wrong command';
	RETURN;
END_CASE

// Send robot target area data
_DO3.nArea1 := _Area.BitList.Bit0;
_DO3.nArea2 := _Area.BitList.Bit1;
_DO3.nArea3 := _Area.BitList.Bit2;
_DO3.nArea4 := _Area.BitList.Bit3;

// Send robot target address data
_DO3.nAddress1 := _Address.BitList.Bit0;
_DO3.nAddress2 := _Address.BitList.Bit1;
_DO3.nAddress3 := _Address.BitList.Bit2;
_DO3.nAddress4 := _Address.BitList.Bit3;
_DO3.nAddress5 := _Address.BitList.Bit4;
_DO3.nAddress6 := _Address.BitList.Bit5;
_DO3.nAddress7 := _Address.BitList.Bit6;


_DO3.bExecute := NOT Error;

_DO3.bContinue := BoxReady;

M_StartAbsMoveAction_ClampA := NOT Error; // Method end
END_METHOD

(* This Method is used to send command data to Fanuc Robot, only clampB is work 
*)
METHOD M_StartAbsMoveAction_ClampB : BOOL
VAR_INPUT
    TargetArea    : E_RobotArea;    // Select the zone where robot will going.
    TargetAddress : E_RobotAddress; // Because the address num in different zone, the number define is different. But also need >= 1, 0 = undefined
    ClampAction   : E_ClampAction;  // need to define the command
    BoxReady      : BOOL;           // Fanuc robot prog will stop at a safe position just before reaching the target location, until `AllowContinue` is set to true.
END_VAR

VAR_OUTPUT
    Error  : BOOL;
    ErrMsg : T_MaxString;
END_VAR

VAR_INST
    _Area    : ST_IntToBool;
    _Address : ST_IntToBool;
END_VAR
// Set target area
_Area.nInt := TargetArea;

// Check ClampB target area is correct
CASE TargetArea OF
    E_RobotArea.RoundBelt..E_RobotArea.PullOutConveyor:
        _Area.nInt := TargetArea;
ELSE
    Error  := TRUE;
    ErrMsg := 'ClampB target area out of range';
	RETURN;
END_CASE

// Check ClampB target address is correct
CASE TargetAddress OF
	E_RobotAddress.Address01..E_RobotAddress.Address06:
		_Address.nInt := TargetAddress;
ELSE
	Error := TRUE;
	ErrMsg := 'ClampB target address is out of range';
	RETURN;
END_CASE

// Check ClampB Action is correct
CASE ClampAction OF
	E_ClampAction.PickUp:
		_DO4.bGet := TRUE;
	E_ClampAction.Place:
		_DO4.bGet := FALSE;
ELSE
	Error := TRUE;
	ErrMsg := 'ClampB Action is wrong command';
	RETURN;
END_CASE

// Send robot target area data
_DO4.nArea1 := _Area.BitList.Bit0;
_DO4.nArea2 := _Area.BitList.Bit1;
_DO4.nArea3 := _Area.BitList.Bit2;
_DO4.nArea4 := _Area.BitList.Bit3;

// Send robot target address data
_DO4.nAddress1 := _Address.BitList.Bit0;
_DO4.nAddress2 := _Address.BitList.Bit1;
_DO4.nAddress3 := _Address.BitList.Bit2;
_DO4.nAddress4 := _Address.BitList.Bit3;
_DO4.nAddress5 := _Address.BitList.Bit4;
_DO4.nAddress6 := _Address.BitList.Bit5;
_DO4.nAddress7 := _Address.BitList.Bit6;

_DO4.bExecute := NOT Error;

_DO4.bContinue := BoxReady;

M_StartAbsMoveAction_ClampB := NOT Error; // Method end
END_METHOD

METHOD M_StartAbsMoveAction_ClampBoth : BOOL
VAR_INPUT
    ClampA_TargetArea    : E_RobotArea;
    ClampA_TargetAddress : E_RobotAddress;
    ClampA_Action        : E_ClampAction;
    ClampB_TargetArea    : E_RobotArea;
    ClampB_TargetAddress : E_RobotAddress;
    ClampB_Action        : E_ClampAction;
    BoxReady_1st         : BOOL;
    BoxReady_2nd         : BOOL;
END_VAR

VAR_OUTPUT
    Error  : BOOL;
    ErrMsg : T_MaxString;
END_VAR

VAR_INST
    _ClampA_Area    : ST_IntToBool;
    _ClampB_Area    : ST_IntToBool;
    _ClampA_Address : ST_IntToBool;
    _ClampB_Address : ST_IntToBool;
END_VAR
// Set Target Area
_ClampA_Area.nInt := ClampA_TargetArea;
_ClampB_Area.nInt := ClampB_TargetArea;
// Check ClampA target area is correct
CASE ClampA_TargetArea OF
    E_RobotArea.RoundBelt..E_RobotArea.PullOutConveyor:
        _ClampA_Area.nInt := ClampA_TargetArea;
ELSE
    Error  := TRUE;
    ErrMsg := 'ClampA target area out of range';
	RETURN;
END_CASE
// Check ClampA target address is correct
CASE ClampA_TargetAddress OF
    E_RobotAddress.Address01..E_RobotAddress.Address06:
        _ClampA_Address.nInt := ClampA_TargetAddress;
ELSE
    Error  := TRUE;
    ErrMsg := 'ClampA target address out of range';
	RETURN;
END_CASE

// Check ClampA Action is correct
CASE ClampA_Action OF
	E_ClampAction.PickUp:
		_DO3.bGet := TRUE;
	E_ClampAction.Place:
		_DO3.bGet := FALSE;
ELSE
	Error := TRUE;
	ErrMsg := 'ClampA Action is wrong command';
	RETURN;
END_CASE
// Check ClampB target area is correct
CASE ClampB_TargetArea OF
    E_RobotArea.RoundBelt..E_RobotArea.PullOutConveyor:
        _ClampB_Area.nInt := ClampB_TargetArea;
ELSE
	Error := TRUE;
	ErrMsg := 'ClampB target area out of range';
	RETURN;
END_CASE

// Check ClampB target address is correct
CASE ClampB_TargetAddress OF
	E_RobotAddress.Address01..E_RobotAddress.Address06:
		_ClampB_Address.nInt := ClampB_TargetAddress;
ELSE
	Error := TRUE;
	ErrMsg := 'ClampB target address is out of range';
	RETURN;
END_CASE
// Check ClampB Action is correct
CASE ClampB_Action OF
	E_ClampAction.PickUp:
		_DO4.bGet := TRUE;
	E_ClampAction.Place:
		_DO4.bGet := FALSE;
ELSE
	Error := TRUE;
	ErrMsg := 'ClampB Action is wrong command';
	RETURN;
END_CASE

// Send robot target area data
_DO3.nArea1 := _ClampA_Area.BitList.Bit0;
_DO3.nArea2 := _ClampA_Area.BitList.Bit1;
_DO3.nArea3 := _ClampA_Area.BitList.Bit2;
_DO3.nArea4 := _ClampA_Area.BitList.Bit3;

_DO4.nArea1 := _ClampB_Area.BitList.Bit0;
_DO4.nArea2 := _ClampB_Area.BitList.Bit1;
_DO4.nArea3 := _ClampB_Area.BitList.Bit2;
_DO4.nArea4 := _ClampB_Area.BitList.Bit3;

// Send robot target address data
_DO3.nAddress1 := _ClampA_Address.BitList.Bit0;
_DO3.nAddress2 := _ClampA_Address.BitList.Bit1;
_DO3.nAddress3 := _ClampA_Address.BitList.Bit2;
_DO3.nAddress4 := _ClampA_Address.BitList.Bit3;
_DO3.nAddress5 := _ClampA_Address.BitList.Bit4;
_DO3.nAddress6 := _ClampA_Address.BitList.Bit5;
_DO3.nAddress7 := _ClampA_Address.BitList.Bit6;

_DO4.nAddress1 := _ClampB_Address.BitList.Bit0;
_DO4.nAddress2 := _ClampB_Address.BitList.Bit1;
_DO4.nAddress3 := _ClampB_Address.BitList.Bit2;
_DO4.nAddress4 := _ClampB_Address.BitList.Bit3;
_DO4.nAddress5 := _ClampB_Address.BitList.Bit4;
_DO4.nAddress6 := _ClampB_Address.BitList.Bit5;
_DO4.nAddress7 := _ClampB_Address.BitList.Bit6;

_DO3.bExecute := NOT Error;
_DO4.bExecute := NOT Error;

_DO3.bContinue := BoxReady_1st;
_DO4.bContinue := BoxReady_2nd;

M_StartAbsMoveAction_ClampBoth := NOT Error; // Method end
END_METHOD

METHOD M_StartMoveBoxToFeedInConveyor_ClampA : BOOL
VAR_INPUT
    ConveyorSlideSelect : E_FeedInEmptyBox_PlaceArea;
    DiffSizeSlideClear  : BOOL;
    SameSizeSlideClear  : BOOL;
END_VAR
VAR_INST
    _Area    : ST_IntToBool;
    _Address : ST_IntToBool;
END_VAR
// Set target area is round belt
_Area.nInt := E_RobotArea.TransmitCV;
IF ConveyorSlideSelect = E_FeedInEmptyBox_PlaceArea.DiffSizeConveyor THEN
	_Address.nInt := 1;
ELSIF ConveyorSlideSelect = E_FeedInEmptyBox_PlaceArea.SameSizeConveyor THEN
	_Address.nInt := 2;
ELSE
	// Wrong command, return
	RETURN ;
END_IF
// Send robot target area data
_DO3.nArea1 := _Area.BitList.Bit0;
_DO3.nArea2 := _Area.BitList.Bit1;
_DO3.nArea3 := _Area.BitList.Bit2;
_DO3.nArea4 := _Area.BitList.Bit3;

// Send robot target address data
_DO3.nAddress1 := _Address.BitList.Bit0;
_DO3.nAddress2 := _Address.BitList.Bit1;
_DO3.nAddress3 := _Address.BitList.Bit2;
_DO3.nAddress4 := _Address.BitList.Bit3;
_DO3.nAddress5 := _Address.BitList.Bit4;
_DO3.nAddress6 := _Address.BitList.Bit5;
_DO3.nAddress7 := _Address.BitList.Bit6;

_DO3.bGet := FALSE; // Place action

_DO3.bExecute := TRUE;
IF ConveyorSlideSelect = E_FeedInEmptyBox_PlaceArea.DiffSizeConveyor THEN
	_DO3.bContinue := DiffSizeSlideClear;
ELSIF ConveyorSlideSelect = E_FeedInEmptyBox_PlaceArea.SameSizeConveyor THEN
	_DO3.bContinue := SameSizeSlideClear;
END_IF
M_StartMoveBoxToFeedInConveyor_ClampA := TRUE ; // Method end
END_METHOD

METHOD M_StartMoveBoxToFeedInConveyor_ClampB : BOOL
VAR_INPUT
	ConveyorSlideSelect : E_FeedInEmptyBox_PlaceArea;
    DiffSizeSlideClear  : BOOL;
    SameSizeSlideClear  : BOOL;
END_VAR
VAR_INST
	_Area : ST_IntToBool;
	_Address_ClampB :ST_IntToBool;
END_VAR
// Set target area is round belt
_Area.nInt := E_RobotArea.TransmitCV;
IF ConveyorSlideSelect = E_FeedInEmptyBox_PlaceArea.DiffSizeConveyor THEN
	_Address_ClampB.nInt := 1;
ELSIF ConveyorSlideSelect = E_FeedInEmptyBox_PlaceArea.SameSizeConveyor THEN
	_Address_ClampB.nInt := 2;
ELSE
	// Wrong command, return
	RETURN ;
END_IF
// Send robot target area data
_DO4.nArea1 := _Area.BitList.Bit0;
_DO4.nArea2 := _Area.BitList.Bit1;
_DO4.nArea3 := _Area.BitList.Bit2;
_DO4.nArea4 := _Area.BitList.Bit3;

// Send robot target address data
_DO4.nAddress1 := _Address_ClampB.BitList.Bit0;
_DO4.nAddress2 := _Address_ClampB.BitList.Bit1;
_DO4.nAddress3 := _Address_ClampB.BitList.Bit2;
_DO4.nAddress4 := _Address_ClampB.BitList.Bit3;
_DO4.nAddress5 := _Address_ClampB.BitList.Bit4;
_DO4.nAddress6 := _Address_ClampB.BitList.Bit5;
_DO4.nAddress7 := _Address_ClampB.BitList.Bit6;

_DO4.bGet := FALSE; // Place action

_DO4.bExecute := TRUE;
IF ConveyorSlideSelect = E_FeedInEmptyBox_PlaceArea.DiffSizeConveyor THEN
	_DO4.bContinue := DiffSizeSlideClear;
ELSIF ConveyorSlideSelect = E_FeedInEmptyBox_PlaceArea.SameSizeConveyor THEN
	_DO4.bContinue := SameSizeSlideClear;
END_IF
M_StartMoveBoxToFeedInConveyor_ClampB := TRUE; // Method end
END_METHOD

METHOD M_StartMoveBoxToFeedInConveyor_ClampBoth : BOOL
VAR_INPUT
//    ConveyorSlideSelect : E_FeedInEmptyBox_PlaceArea;
    ClampA_Address      : E_FeedInEmptyBox_PlaceArea;
    ClampB_Address      : E_FeedInEmptyBox_PlaceArea;
	SlideClear_1st : BOOL;
	SlideClear_2nd : BOOL;
END_VAR
VAR_INST
    _Area           : ST_IntToBool;
    _Address_ClampA : ST_IntToBool;
    _Address_ClampB : ST_IntToBool;
END_VAR
// Set target area is round belt
_Area.nInt := E_RobotArea.TransmitCV;
// Select ClampA target address
IF ClampA_Address = E_FeedInEmptyBox_PlaceArea.DiffSizeConveyor THEN
	_Address_ClampA.nInt := 1;
ELSIF ClampA_Address = E_FeedInEmptyBox_PlaceArea.SameSizeConveyor THEN
	_Address_ClampA.nInt := 2;
ELSE
	// Wrong command, return
	RETURN ;
END_IF

// Select ClampB target address
IF ClampB_Address = E_FeedInEmptyBox_PlaceArea.DiffSizeConveyor THEN
	_Address_ClampB.nInt := 1;
ELSIF ClampB_Address = E_FeedInEmptyBox_PlaceArea.SameSizeConveyor THEN
	_Address_ClampB.nInt := 2;
ELSE
	// Wrong command, return
	RETURN;
END_IF

// Send robot target area data
_DO3.nArea1 := _Area.BitList.Bit0;
_DO3.nArea2 := _Area.BitList.Bit1;
_DO3.nArea3 := _Area.BitList.Bit2;
_DO3.nArea4 := _Area.BitList.Bit3;

_DO4.nArea1 := _Area.BitList.Bit0;
_DO4.nArea2 := _Area.BitList.Bit1;
_DO4.nArea3 := _Area.BitList.Bit2;
_DO4.nArea4 := _Area.BitList.Bit3;

// Send robot clampA target address data
_DO3.nAddress1 := _Address_ClampA.BitList.Bit0;
_DO3.nAddress2 := _Address_ClampA.BitList.Bit1;
_DO3.nAddress3 := _Address_ClampA.BitList.Bit2;
_DO3.nAddress4 := _Address_ClampA.BitList.Bit3;
_DO3.nAddress5 := _Address_ClampA.BitList.Bit4;
_DO3.nAddress6 := _Address_ClampA.BitList.Bit5;
_DO3.nAddress7 := _Address_ClampA.BitList.Bit6;

_do4.nAddress1 := _Address_ClampB.BitList.Bit0;
_do4.nAddress2 := _Address_ClampB.BitList.Bit1;
_do4.nAddress3 := _Address_ClampB.BitList.Bit2;
_do4.nAddress4 := _Address_ClampB.BitList.Bit3;
_do4.nAddress5 := _Address_ClampB.BitList.Bit4;
_do4.nAddress6 := _Address_ClampB.BitList.Bit5;
_do4.nAddress7 := _Address_ClampB.BitList.Bit6;


_DO3.bGet := FALSE;
_DO4.bGet := FALSE;

_DO3.bExecute := TRUE;
_DO4.bExecute := TRUE;

_DO3.bContinue := SlideClear_1st;
_DO4.bContinue := SlideClear_2nd;

M_StartMoveBoxToFeedInConveyor_ClampBoth := TRUE; // Method end
END_METHOD

METHOD M_StartMoveBoxToRoundBelt_Both : BOOL
VAR_INPUT
	CarrierSelect_ClampA : E_ReloadRoundBelt_PlaceAddress;
	CarrierSelect_ClampB : E_ReloadRoundBelt_PlaceAddress;
	A2_Sensor : BOOL;
	A3_Sensor : BOOL;
	RoundBeltSafe_1st : BOOL;
	RoundBeltSafe_2nd : BOOL;
END_VAR
VAR_INST
	_Area1 : ST_IntToBool;
	_Address1 : ST_IntToBool;
	CarrierAddress1 :E_ReloadRoundBelt_PlaceAddress;
	_Area2: ST_IntToBool;
	_Address2 : ST_IntToBool;
	CarrierAddress2 :E_ReloadRoundBelt_PlaceAddress;
END_VAR
// Set target area is round belt
_Area1.nInt := E_RobotArea.RoundBelt;
_Area2.nInt := E_RobotArea.RoundBelt;

IF CarrierSelect_ClampA = E_ReloadRoundBelt_PlaceAddress.A2 THEN
	_Address1.nInt := 1;
ELSIF CarrierSelect_ClampA = E_ReloadRoundBelt_PlaceAddress.A3 THEN
	_Address1.nInt := 2;
ELSE
	// Wrong command, return
	RETURN;
END_IF

IF CarrierSelect_ClampB = E_ReloadRoundBelt_PlaceAddress.A2 THEN
	_Address2.nInt := 1;
ELSIF CarrierSelect_ClampB = E_ReloadRoundBelt_PlaceAddress.A3 THEN
	_Address2.nInt := 2;
ELSE
	// Wrong command return
	RETURN;
END_IF
// Send robot target area data
_DO3.nArea1 := _Area1.BitList.Bit0;
_DO3.nArea2 := _Area1.BitList.Bit1;
_DO3.nArea3 := _Area1.BitList.Bit2;
_DO3.nArea4 := _Area1.BitList.Bit3;

_DO4.nArea1 := _Area2.BitList.Bit0;
_DO4.nArea2 := _Area2.BitList.Bit1;
_DO4.nArea3 := _Area2.BitList.Bit2;
_DO4.nArea4 := _Area2.BitList.Bit3;

// Send robot target address data
_DO3.nAddress1 := _Address1.BitList.Bit0;
_DO3.nAddress2 := _Address1.BitList.Bit1;
_DO3.nAddress3 := _Address1.BitList.Bit2;
_DO3.nAddress4 := _Address1.BitList.Bit3;
_DO3.nAddress5 := _Address1.BitList.Bit4;
_DO3.nAddress6 := _Address1.BitList.Bit5;
_DO3.nAddress7 := _Address1.BitList.Bit6;

_DO4.nAddress1 := _Address2.BitList.Bit0;
_DO4.nAddress2 := _Address2.BitList.Bit1;
_DO4.nAddress3 := _Address2.BitList.Bit2;
_DO4.nAddress4 := _Address2.BitList.Bit3;
_DO4.nAddress5 := _Address2.BitList.Bit4;
_DO4.nAddress6 := _Address2.BitList.Bit5;
_DO4.nAddress7 := _Address2.BitList.Bit6;

_DO3.bGet := FALSE; // ClampA Place action
_DO4.bGet := FALSE; // ClampB Place action

IF CarrierSelect_ClampA = E_ReloadRoundBelt_PlaceAddress.A2 THEN
	_DO3.bContinue := NOT A2_Sensor AND RoundBeltSafe_1st;
ELSIF 	CarrierSelect_ClampA = E_ReloadRoundBelt_PlaceAddress.A3 THEN
	_DO3.bContinue := NOT A3_Sensor AND RoundBeltSafe_1st;
END_IF

IF CarrierSelect_ClampB = E_ReloadRoundBelt_PlaceAddress.A2 THEN
	_DO4.bContinue := NOT A2_Sensor AND RoundBeltSafe_2nd;
ELSIF CarrierSelect_ClampB = E_ReloadRoundBelt_PlaceAddress.A3 THEN
	_DO4.bContinue := NOT A3_Sensor AND RoundBeltSafe_2nd;
END_IF

_DO3.bExecute := TRUE; // ClampA Place action
_DO4.bExecute := TRUE; // ClampB Place action


M_StartMoveBoxToRoundBelt_Both := TRUE; // Method end
END_METHOD

METHOD M_StartMoveBoxToRoundBelt_ClampA : BOOL
VAR_INPUT
    CarrierSelect : E_ReloadRoundBelt_PlaceAddress;
    A2_Sensor     : BOOL;
    A3_Sensor     : BOOL;
	RoundBeltSafe : BOOL;
END_VAR
VAR_INST
    _Area          : ST_IntToBool;
    _Address       : ST_IntToBool;
    CarrierAddress : E_ReloadRoundBelt_PlaceAddress;
END_VAR
// Set target area is round belt
_Area.nInt := E_RobotArea.RoundBelt;

IF CarrierSelect = E_ReloadRoundBelt_PlaceAddress.A2 THEN
    _Address.nInt := 1;
ELSIF CarrierSelect = E_ReloadRoundBelt_PlaceAddress.A3 THEN
    _Address.nInt := 2;
ELSE
    // Wrong command, return
    RETURN;
END_IF

// Send robot target area data
_DO3.nArea1 := _Area.BitList.Bit0;
_DO3.nArea2 := _Area.BitList.Bit1;
_DO3.nArea3 := _Area.BitList.Bit2;
_DO3.nArea4 := _Area.BitList.Bit3;

// Send robot target address data
_DO3.nAddress1 := _Address.BitList.Bit0;
_DO3.nAddress2 := _Address.BitList.Bit1;
_DO3.nAddress3 := _Address.BitList.Bit2;
_DO3.nAddress4 := _Address.BitList.Bit3;
_DO3.nAddress5 := _Address.BitList.Bit4;
_DO3.nAddress6 := _Address.BitList.Bit5;
_DO3.nAddress7 := _Address.BitList.Bit6;

_DO3.bGet := FALSE; // Place action

_DO3.bExecute := TRUE;

IF CarrierSelect = E_ReloadRoundBelt_PlaceAddress.A2 THEN
    _DO3.bContinue := NOT A2_Sensor AND RoundBeltSafe ; // Carrier A2 did not has box
ELSIF CarrierSelect = E_ReloadRoundBelt_PlaceAddress.A3 THEN
    _DO3.bContinue := NOT A3_Sensor AND RoundBeltSafe; // Carrier A3 did not has box
END_IF

M_StartMoveBoxToRoundBelt_ClampA := true; // Method end
END_METHOD

METHOD M_StartMoveBoxToRoundBelt_ClampB : BOOL
VAR_INPUT
    CarrierSelect : E_ReloadRoundBelt_PlaceAddress;
    A2_Sensor     : BOOL;
    A3_Sensor     : BOOL;
	RoundBeltSafe : BOOL;
END_VAR
VAR_INST
    _Area          : ST_IntToBool;
    _Address       : ST_IntToBool;
    CarrierAddress : E_ReloadRoundBelt_PlaceAddress;
END_VAR
// Set target area is round belt
_Area.nInt := E_RobotArea.RoundBelt;
IF CarrierSelect = E_ReloadRoundBelt_PlaceAddress.A2 THEN
	_Address.nInt := 1;
ELSIF  CarrierSelect = E_ReloadRoundBelt_PlaceAddress.A3 THEN
	_Address.nInt := 2;
ELSE
	// Wrong command, return
	RETURN ;
END_IF

// Send robot target area data
_DO4.nArea1 := _Area.BitList.Bit0;
_DO4.nArea2 := _Area.BitList.Bit1;
_DO4.nArea3 := _Area.BitList.Bit2;
_DO4.nArea4 := _Area.BitList.Bit3;

// Send robot target address data
_DO4.nAddress1 := _Address.BitList.Bit0;
_DO4.nAddress2 := _Address.BitList.Bit1;
_DO4.nAddress3 := _Address.BitList.Bit2;
_DO4.nAddress4 := _Address.BitList.Bit3;
_DO4.nAddress5 := _Address.BitList.Bit4;
_DO4.nAddress6 := _Address.BitList.Bit5;
_DO4.nAddress7 := _Address.BitList.Bit6;

_DO4.bGet := FALSE; // Place action

_DO4.bExecute := TRUE;

IF CarrierSelect = E_ReloadRoundBelt_PlaceAddress.A2 THEN
	_DO4.bContinue := NOT A2_Sensor AND RoundBeltSafe; // Carrier A2 did not has box
ELSIF CarrierSelect = E_ReloadRoundBelt_PlaceAddress.A3 THEN
	_DO4.bContinue := NOT A3_Sensor AND RoundBeltSafe; // Carrier A3 did not has box
END_IF

